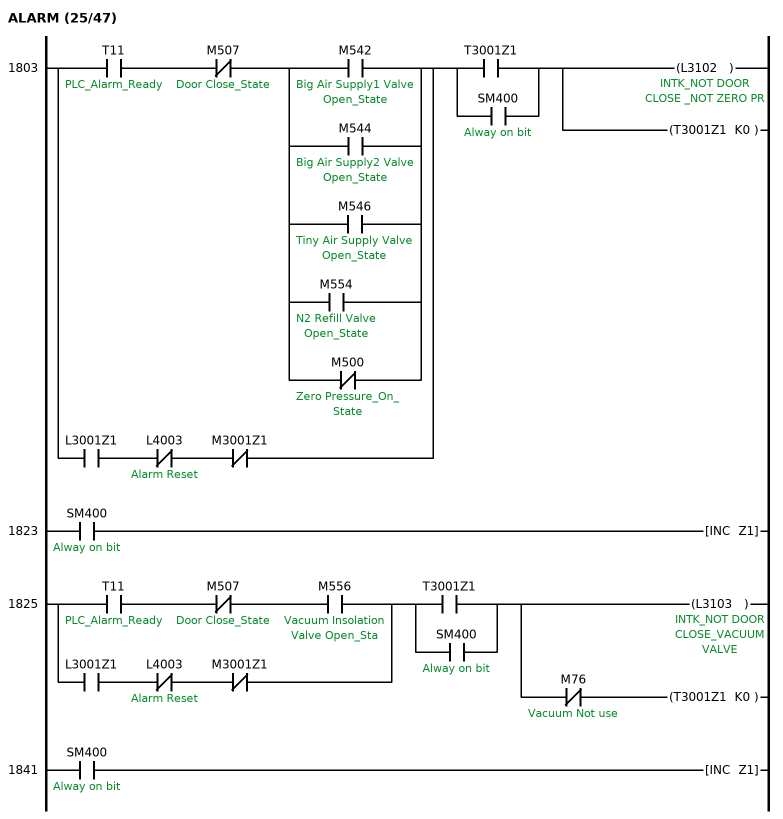
1803  LD      T11  ; PLC_Alarm_Ready
      ANI     M507  ; Door Close_State
      LD      M542  ; Big Air Supply1 Valve Open_State
      OR      M544  ; Big Air Supply2 Valve Open_State
      OR      M546  ; Tiny Air Supply Valve Open_State
      OR      M554  ; N2 Refill Valve Open_State
      ORI     M500  ; Zero Pressure_On_State
      ANB
      LD      L3001Z1
      ANI     L4003  ; Alarm Reset
      ANI     M3001Z1
      ORB
      LD      T3001Z1
      OR      SM400  ; Alway on bit
      ANB
      OUT     L3102  ; INTK_NOT DOOR CLOSE _NOT ZERO PR
      OUT     T3001Z1 K0
1823  LD      SM400  ; Alway on bit
      INC     Z1
1825  LD      T11  ; PLC_Alarm_Ready
      ANI     M507  ; Door Close_State
      AND     M556  ; Vacuum Insolation Valve Open_Sta
      LD      L3001Z1
      ANI     L4003  ; Alarm Reset
      ANI     M3001Z1
      ORB
      LD      T3001Z1
      OR      SM400  ; Alway on bit
      ANB
      OUT     L3103  ; INTK_NOT DOOR CLOSE_VACUUM VALVE
      ANI     M76  ; Vacuum Not use
      OUT     T3001Z1 K0
1841  LD      SM400  ; Alway on bit
      INC     Z1
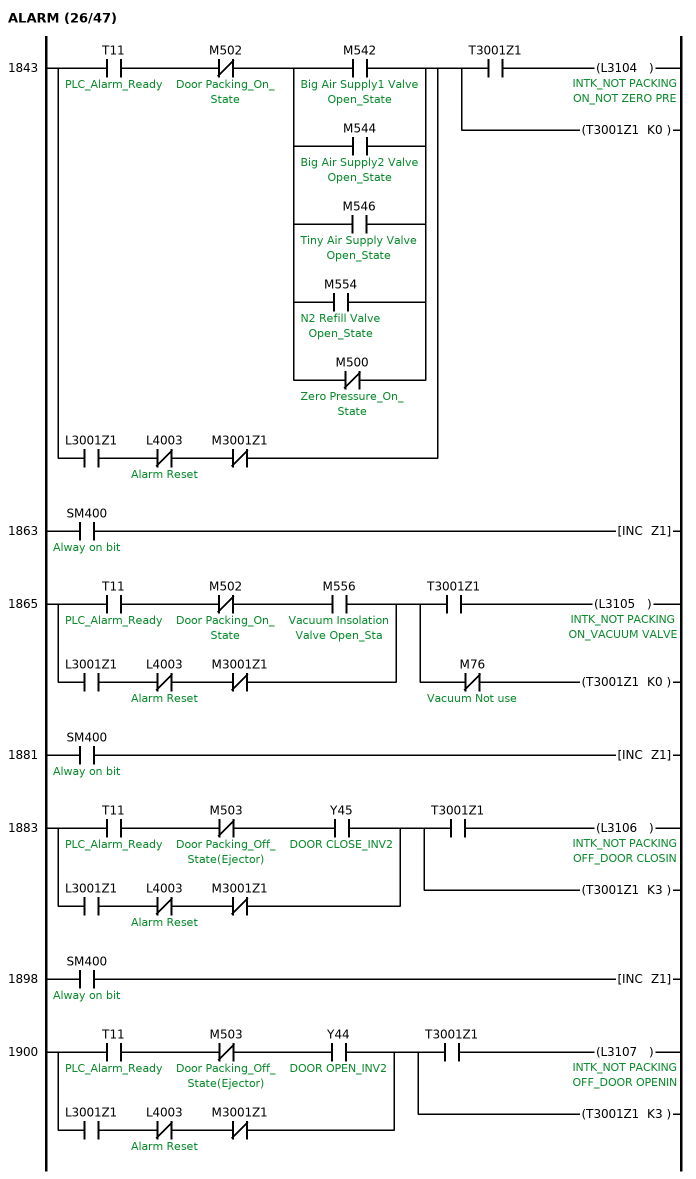
1843  LD      T11  ; PLC_Alarm_Ready
      ANI     M502  ; Door Packing_On_State
      LD      M542  ; Big Air Supply1 Valve Open_State
      OR      M544  ; Big Air Supply2 Valve Open_State
      OR      M546  ; Tiny Air Supply Valve Open_State
      OR      M554  ; N2 Refill Valve Open_State
      ORI     M500  ; Zero Pressure_On_State
      ANB
      LD      L3001Z1
      ANI     L4003  ; Alarm Reset
      ANI     M3001Z1
      ORB
      MPS
      AND     T3001Z1
      OUT     L3104  ; INTK_NOT PACKING ON_NOT ZERO PRE
      MPP
      OUT     T3001Z1 K0
1863  LD      SM400  ; Alway on bit
      INC     Z1
1865  LD      T11  ; PLC_Alarm_Ready
      ANI     M502  ; Door Packing_On_State
      AND     M556  ; Vacuum Insolation Valve Open_Sta
      LD      L3001Z1
      ANI     L4003  ; Alarm Reset
      ANI     M3001Z1
      ORB
      MPS
      AND     T3001Z1
      OUT     L3105  ; INTK_NOT PACKING ON_VACUUM VALVE
      MPP
      ANI     M76  ; Vacuum Not use
      OUT     T3001Z1 K0
1881  LD      SM400  ; Alway on bit
      INC     Z1
1883  LD      T11  ; PLC_Alarm_Ready
      ANI     M503  ; Door Packing_Off_State(Ejector)
      AND     Y45  ; DOOR CLOSE_INV2
      LD      L3001Z1
      ANI     L4003  ; Alarm Reset
      ANI     M3001Z1
      ORB
      MPS
      AND     T3001Z1
      OUT     L3106  ; INTK_NOT PACKING OFF_DOOR CLOSIN
      MPP
      OUT     T3001Z1 K3
1898  LD      SM400  ; Alway on bit
      INC     Z1
1900  LD      T11  ; PLC_Alarm_Ready
      ANI     M503  ; Door Packing_Off_State(Ejector)
      AND     Y44  ; DOOR OPEN_INV2
      LD      L3001Z1
      ANI     L4003  ; Alarm Reset
      ANI     M3001Z1
      ORB
      MPS
      AND     T3001Z1
      OUT     L3107  ; INTK_NOT PACKING OFF_DOOR OPENIN
      MPP
      OUT     T3001Z1 K3
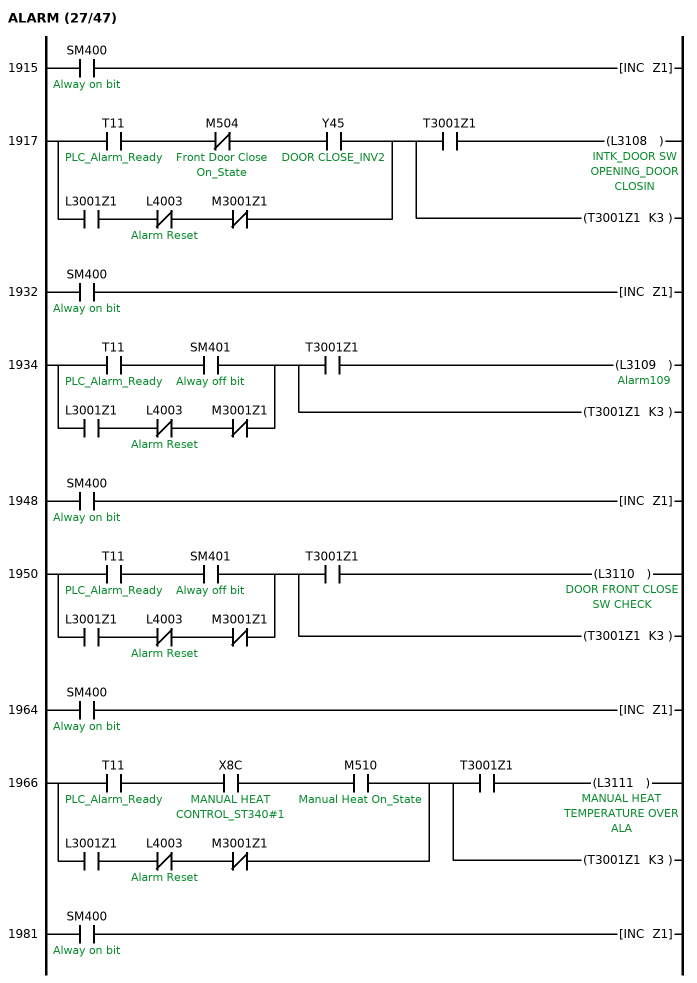
1915  LD      SM400  ; Alway on bit
      INC     Z1
1917  LD      T11  ; PLC_Alarm_Ready
      ANI     M504  ; Front Door Close On_State
      AND     Y45  ; DOOR CLOSE_INV2
      LD      L3001Z1
      ANI     L4003  ; Alarm Reset
      ANI     M3001Z1
      ORB
      MPS
      AND     T3001Z1
      OUT     L3108  ; INTK_DOOR SW OPENING_DOOR CLOSIN
      MPP
      OUT     T3001Z1 K3
1932  LD      SM400  ; Alway on bit
      INC     Z1
1934  LD      T11  ; PLC_Alarm_Ready
      AND     SM401  ; Alway off bit
      LD      L3001Z1
      ANI     L4003  ; Alarm Reset
      ANI     M3001Z1
      ORB
      MPS
      AND     T3001Z1
      OUT     L3109  ; Alarm109
      MPP
      OUT     T3001Z1 K3
1948  LD      SM400  ; Alway on bit
      INC     Z1
1950  LD      T11  ; PLC_Alarm_Ready
      AND     SM401  ; Alway off bit
      LD      L3001Z1
      ANI     L4003  ; Alarm Reset
      ANI     M3001Z1
      ORB
      MPS
      AND     T3001Z1
      OUT     L3110  ; DOOR FRONT CLOSE SW CHECK
      MPP
      OUT     T3001Z1 K3
1964  LD      SM400  ; Alway on bit
      INC     Z1
1966  LD      T11  ; PLC_Alarm_Ready
      AND     X8C  ; MANUAL HEAT CONTROL_ST340#1
      AND     M510  ; Manual Heat On_State
      LD      L3001Z1
      ANI     L4003  ; Alarm Reset
      ANI     M3001Z1
      ORB
      MPS
      AND     T3001Z1
      OUT     L3111  ; MANUAL HEAT TEMPERATURE OVER ALA
      MPP
      OUT     T3001Z1 K3
1981  LD      SM400  ; Alway on bit
      INC     Z1
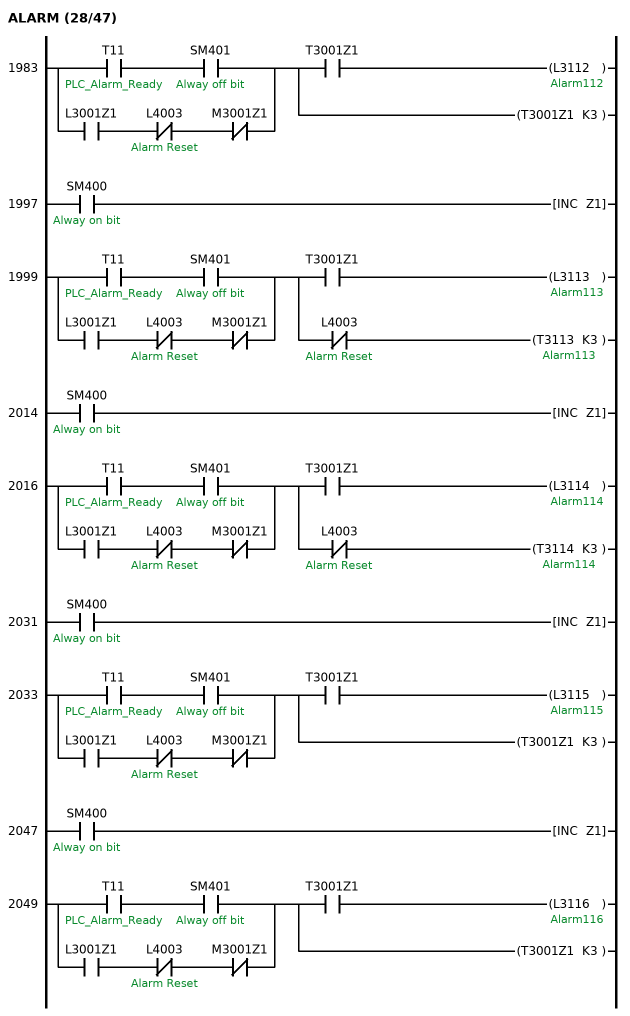
1983  LD      T11  ; PLC_Alarm_Ready
      AND     SM401  ; Alway off bit
      LD      L3001Z1
      ANI     L4003  ; Alarm Reset
      ANI     M3001Z1
      ORB
      MPS
      AND     T3001Z1
      OUT     L3112  ; Alarm112
      MPP
      OUT     T3001Z1 K3
1997  LD      SM400  ; Alway on bit
      INC     Z1
1999  LD      T11  ; PLC_Alarm_Ready
      AND     SM401  ; Alway off bit
      LD      L3001Z1
      ANI     L4003  ; Alarm Reset
      ANI     M3001Z1
      ORB
      MPS
      AND     T3001Z1
      OUT     L3113  ; Alarm113
      MPP
      ANI     L4003  ; Alarm Reset
      OUT     T3113 K3  ; Alarm113
2014  LD      SM400  ; Alway on bit
      INC     Z1
2016  LD      T11  ; PLC_Alarm_Ready
      AND     SM401  ; Alway off bit
      LD      L3001Z1
      ANI     L4003  ; Alarm Reset
      ANI     M3001Z1
      ORB
      MPS
      AND     T3001Z1
      OUT     L3114  ; Alarm114
      MPP
      ANI     L4003  ; Alarm Reset
      OUT     T3114 K3  ; Alarm114
2031  LD      SM400  ; Alway on bit
      INC     Z1
2033  LD      T11  ; PLC_Alarm_Ready
      AND     SM401  ; Alway off bit
      LD      L3001Z1
      ANI     L4003  ; Alarm Reset
      ANI     M3001Z1
      ORB
      MPS
      AND     T3001Z1
      OUT     L3115  ; Alarm115
      MPP
      OUT     T3001Z1 K3
2047  LD      SM400  ; Alway on bit
      INC     Z1
2049  LD      T11  ; PLC_Alarm_Ready
      AND     SM401  ; Alway off bit
      LD      L3001Z1
      ANI     L4003  ; Alarm Reset
      ANI     M3001Z1
      ORB
      MPS
      AND     T3001Z1
      OUT     L3116  ; Alarm116
      MPP
      OUT     T3001Z1 K3
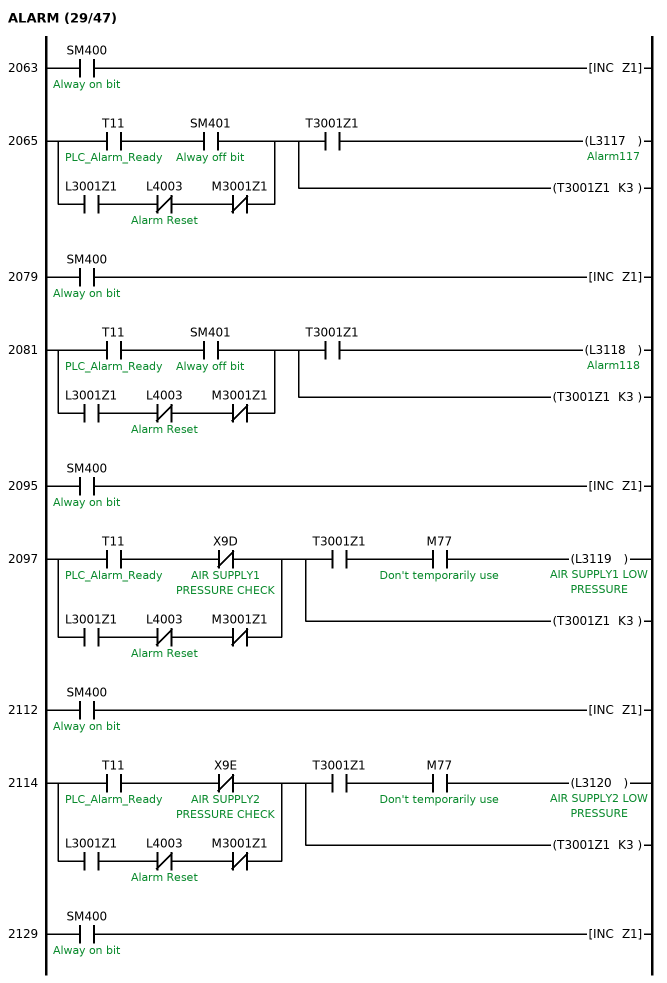
2063  LD      SM400  ; Alway on bit
      INC     Z1
2065  LD      T11  ; PLC_Alarm_Ready
      AND     SM401  ; Alway off bit
      LD      L3001Z1
      ANI     L4003  ; Alarm Reset
      ANI     M3001Z1
      ORB
      MPS
      AND     T3001Z1
      OUT     L3117  ; Alarm117
      MPP
      OUT     T3001Z1 K3
2079  LD      SM400  ; Alway on bit
      INC     Z1
2081  LD      T11  ; PLC_Alarm_Ready
      AND     SM401  ; Alway off bit
      LD      L3001Z1
      ANI     L4003  ; Alarm Reset
      ANI     M3001Z1
      ORB
      MPS
      AND     T3001Z1
      OUT     L3118  ; Alarm118
      MPP
      OUT     T3001Z1 K3
2095  LD      SM400  ; Alway on bit
      INC     Z1
2097  LD      T11  ; PLC_Alarm_Ready
      ANI     X9D  ; AIR SUPPLY1 PRESSURE CHECK
      LD      L3001Z1
      ANI     L4003  ; Alarm Reset
      ANI     M3001Z1
      ORB
      MPS
      AND     T3001Z1
      AND     M77  ; Don't temporarily use
      OUT     L3119  ; AIR SUPPLY1 LOW PRESSURE
      MPP
      OUT     T3001Z1 K3
2112  LD      SM400  ; Alway on bit
      INC     Z1
2114  LD      T11  ; PLC_Alarm_Ready
      ANI     X9E  ; AIR SUPPLY2 PRESSURE CHECK
      LD      L3001Z1
      ANI     L4003  ; Alarm Reset
      ANI     M3001Z1
      ORB
      MPS
      AND     T3001Z1
      AND     M77  ; Don't temporarily use
      OUT     L3120  ; AIR SUPPLY2 LOW PRESSURE
      MPP
      OUT     T3001Z1 K3
2129  LD      SM400  ; Alway on bit
      INC     Z1
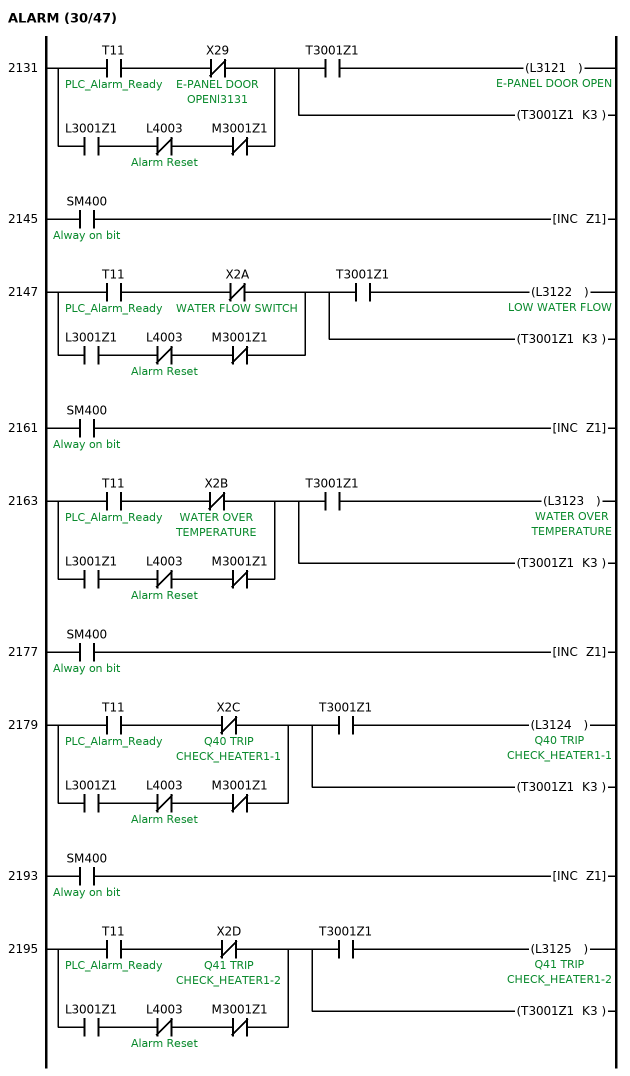
2131  LD      T11  ; PLC_Alarm_Ready
      ANI     X29  ; E-PANEL DOOR OPENl3131
      LD      L3001Z1
      ANI     L4003  ; Alarm Reset
      ANI     M3001Z1
      ORB
      MPS
      AND     T3001Z1
      OUT     L3121  ; E-PANEL DOOR OPEN
      MPP
      OUT     T3001Z1 K3
2145  LD      SM400  ; Alway on bit
      INC     Z1
2147  LD      T11  ; PLC_Alarm_Ready
      ANI     X2A  ; WATER FLOW SWITCH
      LD      L3001Z1
      ANI     L4003  ; Alarm Reset
      ANI     M3001Z1
      ORB
      MPS
      AND     T3001Z1
      OUT     L3122  ; LOW WATER FLOW
      MPP
      OUT     T3001Z1 K3
2161  LD      SM400  ; Alway on bit
      INC     Z1
2163  LD      T11  ; PLC_Alarm_Ready
      ANI     X2B  ; WATER OVER TEMPERATURE
      LD      L3001Z1
      ANI     L4003  ; Alarm Reset
      ANI     M3001Z1
      ORB
      MPS
      AND     T3001Z1
      OUT     L3123  ; WATER OVER TEMPERATURE
      MPP
      OUT     T3001Z1 K3
2177  LD      SM400  ; Alway on bit
      INC     Z1
2179  LD      T11  ; PLC_Alarm_Ready
      ANI     X2C  ; Q40 TRIP CHECK_HEATER1-1
      LD      L3001Z1
      ANI     L4003  ; Alarm Reset
      ANI     M3001Z1
      ORB
      MPS
      AND     T3001Z1
      OUT     L3124  ; Q40 TRIP CHECK_HEATER1-1
      MPP
      OUT     T3001Z1 K3
2193  LD      SM400  ; Alway on bit
      INC     Z1
2195  LD      T11  ; PLC_Alarm_Ready
      ANI     X2D  ; Q41 TRIP CHECK_HEATER1-2
      LD      L3001Z1
      ANI     L4003  ; Alarm Reset
      ANI     M3001Z1
      ORB
      MPS
      AND     T3001Z1
      OUT     L3125  ; Q41 TRIP CHECK_HEATER1-2
      MPP
      OUT     T3001Z1 K3
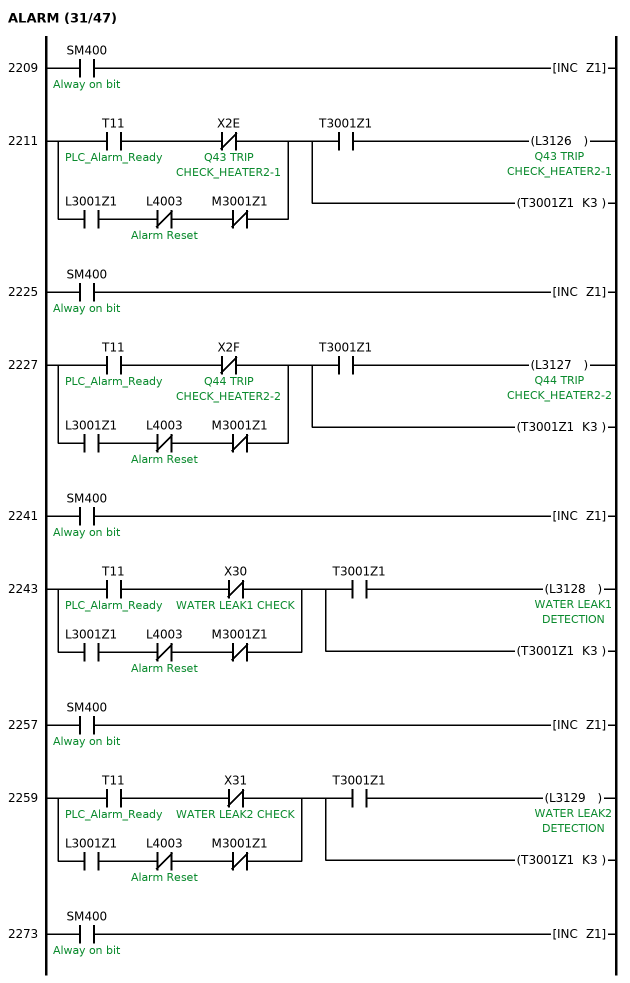
2209  LD      SM400  ; Alway on bit
      INC     Z1
2211  LD      T11  ; PLC_Alarm_Ready
      ANI     X2E  ; Q43 TRIP CHECK_HEATER2-1
      LD      L3001Z1
      ANI     L4003  ; Alarm Reset
      ANI     M3001Z1
      ORB
      MPS
      AND     T3001Z1
      OUT     L3126  ; Q43 TRIP CHECK_HEATER2-1
      MPP
      OUT     T3001Z1 K3
2225  LD      SM400  ; Alway on bit
      INC     Z1
2227  LD      T11  ; PLC_Alarm_Ready
      ANI     X2F  ; Q44 TRIP CHECK_HEATER2-2
      LD      L3001Z1
      ANI     L4003  ; Alarm Reset
      ANI     M3001Z1
      ORB
      MPS
      AND     T3001Z1
      OUT     L3127  ; Q44 TRIP CHECK_HEATER2-2
      MPP
      OUT     T3001Z1 K3
2241  LD      SM400  ; Alway on bit
      INC     Z1
2243  LD      T11  ; PLC_Alarm_Ready
      ANI     X30  ; WATER LEAK1 CHECK
      LD      L3001Z1
      ANI     L4003  ; Alarm Reset
      ANI     M3001Z1
      ORB
      MPS
      AND     T3001Z1
      OUT     L3128  ; WATER LEAK1 DETECTION
      MPP
      OUT     T3001Z1 K3
2257  LD      SM400  ; Alway on bit
      INC     Z1
2259  LD      T11  ; PLC_Alarm_Ready
      ANI     X31  ; WATER LEAK2 CHECK
      LD      L3001Z1
      ANI     L4003  ; Alarm Reset
      ANI     M3001Z1
      ORB
      MPS
      AND     T3001Z1
      OUT     L3129  ; WATER LEAK2 DETECTION
      MPP
      OUT     T3001Z1 K3
2273  LD      SM400  ; Alway on bit
      INC     Z1
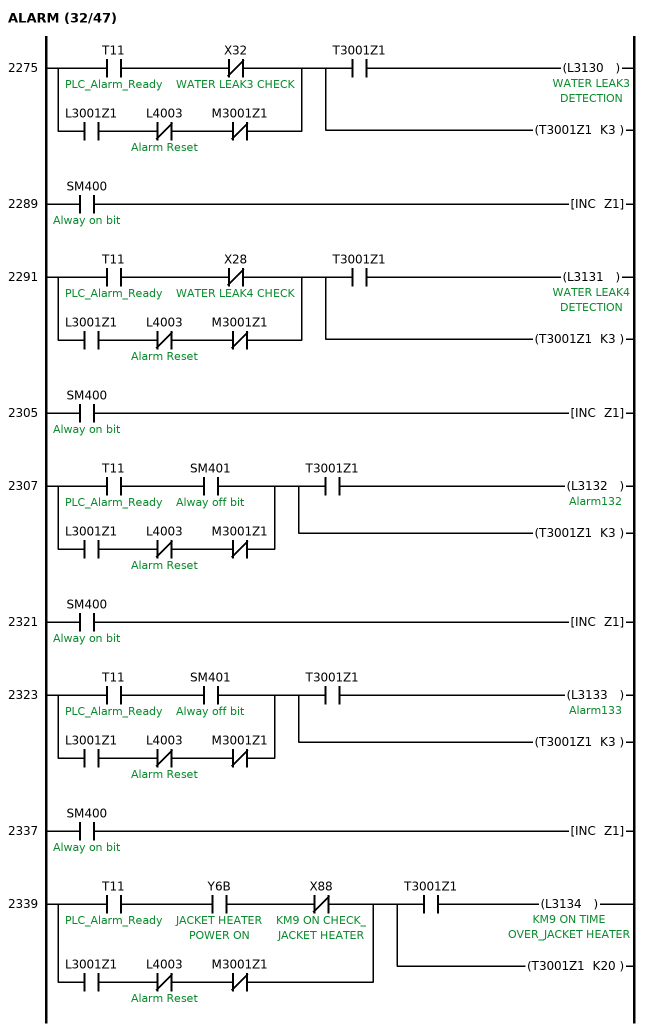
2275  LD      T11  ; PLC_Alarm_Ready
      ANI     X32  ; WATER LEAK3 CHECK
      LD      L3001Z1
      ANI     L4003  ; Alarm Reset
      ANI     M3001Z1
      ORB
      MPS
      AND     T3001Z1
      OUT     L3130  ; WATER LEAK3 DETECTION
      MPP
      OUT     T3001Z1 K3
2289  LD      SM400  ; Alway on bit
      INC     Z1
2291  LD      T11  ; PLC_Alarm_Ready
      ANI     X28  ; WATER LEAK4 CHECK
      LD      L3001Z1
      ANI     L4003  ; Alarm Reset
      ANI     M3001Z1
      ORB
      MPS
      AND     T3001Z1
      OUT     L3131  ; WATER LEAK4 DETECTION
      MPP
      OUT     T3001Z1 K3
2305  LD      SM400  ; Alway on bit
      INC     Z1
2307  LD      T11  ; PLC_Alarm_Ready
      AND     SM401  ; Alway off bit
      LD      L3001Z1
      ANI     L4003  ; Alarm Reset
      ANI     M3001Z1
      ORB
      MPS
      AND     T3001Z1
      OUT     L3132  ; Alarm132
      MPP
      OUT     T3001Z1 K3
2321  LD      SM400  ; Alway on bit
      INC     Z1
2323  LD      T11  ; PLC_Alarm_Ready
      AND     SM401  ; Alway off bit
      LD      L3001Z1
      ANI     L4003  ; Alarm Reset
      ANI     M3001Z1
      ORB
      MPS
      AND     T3001Z1
      OUT     L3133  ; Alarm133
      MPP
      OUT     T3001Z1 K3
2337  LD      SM400  ; Alway on bit
      INC     Z1
2339  LD      T11  ; PLC_Alarm_Ready
      AND     Y6B  ; JACKET HEATER POWER ON
      ANI     X88  ; KM9 ON CHECK_JACKET HEATER
      LD      L3001Z1
      ANI     L4003  ; Alarm Reset
      ANI     M3001Z1
      ORB
      MPS
      AND     T3001Z1
      OUT     L3134  ; KM9 ON TIME OVER_JACKET HEATER
      MPP
      OUT     T3001Z1 K20
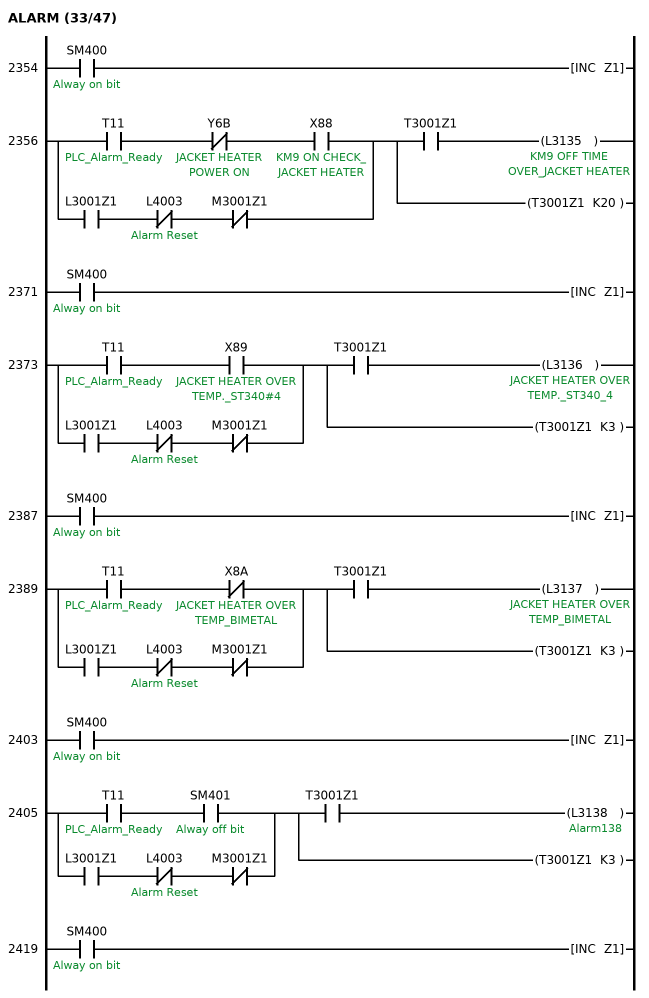
2354  LD      SM400  ; Alway on bit
      INC     Z1
2356  LD      T11  ; PLC_Alarm_Ready
      ANI     Y6B  ; JACKET HEATER POWER ON
      AND     X88  ; KM9 ON CHECK_JACKET HEATER
      LD      L3001Z1
      ANI     L4003  ; Alarm Reset
      ANI     M3001Z1
      ORB
      MPS
      AND     T3001Z1
      OUT     L3135  ; KM9 OFF TIME OVER_JACKET HEATER
      MPP
      OUT     T3001Z1 K20
2371  LD      SM400  ; Alway on bit
      INC     Z1
2373  LD      T11  ; PLC_Alarm_Ready
      AND     X89  ; JACKET HEATER OVER TEMP._ST340#4
      LD      L3001Z1
      ANI     L4003  ; Alarm Reset
      ANI     M3001Z1
      ORB
      MPS
      AND     T3001Z1
      OUT     L3136  ; JACKET HEATER OVER TEMP._ST340_4
      MPP
      OUT     T3001Z1 K3
2387  LD      SM400  ; Alway on bit
      INC     Z1
2389  LD      T11  ; PLC_Alarm_Ready
      ANI     X8A  ; JACKET HEATER OVER TEMP_BIMETAL
      LD      L3001Z1
      ANI     L4003  ; Alarm Reset
      ANI     M3001Z1
      ORB
      MPS
      AND     T3001Z1
      OUT     L3137  ; JACKET HEATER OVER TEMP_BIMETAL
      MPP
      OUT     T3001Z1 K3
2403  LD      SM400  ; Alway on bit
      INC     Z1
2405  LD      T11  ; PLC_Alarm_Ready
      AND     SM401  ; Alway off bit
      LD      L3001Z1
      ANI     L4003  ; Alarm Reset
      ANI     M3001Z1
      ORB
      MPS
      AND     T3001Z1
      OUT     L3138  ; Alarm138
      MPP
      OUT     T3001Z1 K3
2419  LD      SM400  ; Alway on bit
      INC     Z1
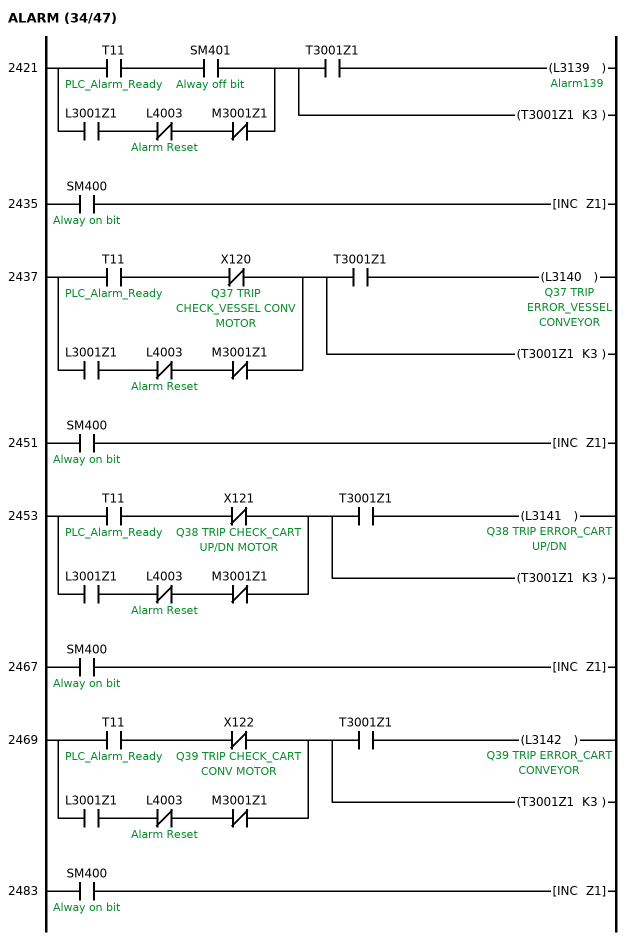
2421  LD      T11  ; PLC_Alarm_Ready
      AND     SM401  ; Alway off bit
      LD      L3001Z1
      ANI     L4003  ; Alarm Reset
      ANI     M3001Z1
      ORB
      MPS
      AND     T3001Z1
      OUT     L3139  ; Alarm139
      MPP
      OUT     T3001Z1 K3
2435  LD      SM400  ; Alway on bit
      INC     Z1
2437  LD      T11  ; PLC_Alarm_Ready
      ANI     X120  ; Q37 TRIP CHECK_VESSEL CONV MOTOR
      LD      L3001Z1
      ANI     L4003  ; Alarm Reset
      ANI     M3001Z1
      ORB
      MPS
      AND     T3001Z1
      OUT     L3140  ; Q37 TRIP ERROR_VESSEL CONVEYOR
      MPP
      OUT     T3001Z1 K3
2451  LD      SM400  ; Alway on bit
      INC     Z1
2453  LD      T11  ; PLC_Alarm_Ready
      ANI     X121  ; Q38 TRIP CHECK_CART UP/DN MOTOR
      LD      L3001Z1
      ANI     L4003  ; Alarm Reset
      ANI     M3001Z1
      ORB
      MPS
      AND     T3001Z1
      OUT     L3141  ; Q38 TRIP ERROR_CART UP/DN
      MPP
      OUT     T3001Z1 K3
2467  LD      SM400  ; Alway on bit
      INC     Z1
2469  LD      T11  ; PLC_Alarm_Ready
      ANI     X122  ; Q39 TRIP CHECK_CART CONV MOTOR
      LD      L3001Z1
      ANI     L4003  ; Alarm Reset
      ANI     M3001Z1
      ORB
      MPS
      AND     T3001Z1
      OUT     L3142  ; Q39 TRIP ERROR_CART CONVEYOR
      MPP
      OUT     T3001Z1 K3
2483  LD      SM400  ; Alway on bit
      INC     Z1
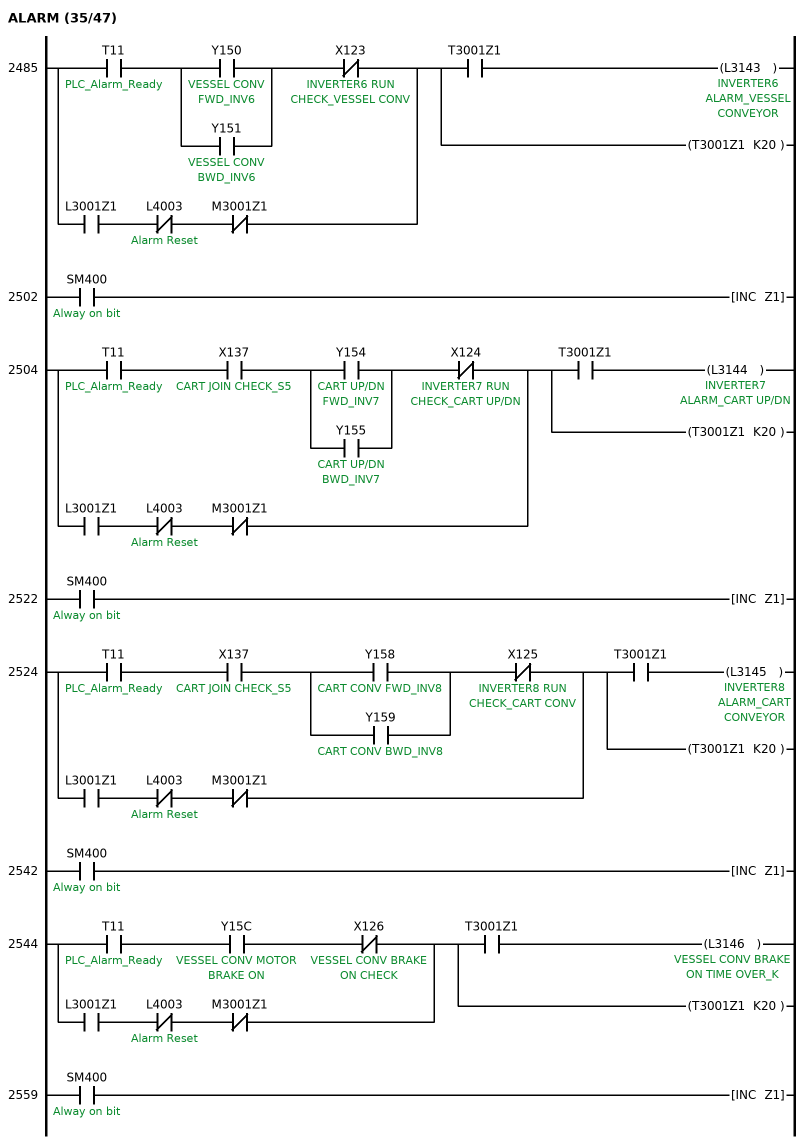
2485  LD      T11  ; PLC_Alarm_Ready
      LD      Y150  ; VESSEL CONV FWD_INV6
      OR      Y151  ; VESSEL CONV BWD_INV6
      ANB
      ANI     X123  ; INVERTER6 RUN CHECK_VESSEL CONV
      LD      L3001Z1
      ANI     L4003  ; Alarm Reset
      ANI     M3001Z1
      ORB
      MPS
      AND     T3001Z1
      OUT     L3143  ; INVERTER6 ALARM_VESSEL CONVEYOR
      MPP
      OUT     T3001Z1 K20
2502  LD      SM400  ; Alway on bit
      INC     Z1
2504  LD      T11  ; PLC_Alarm_Ready
      AND     X137  ; CART JOIN CHECK_S5
      LD      Y154  ; CART UP/DN FWD_INV7
      OR      Y155  ; CART UP/DN BWD_INV7
      ANB
      ANI     X124  ; INVERTER7 RUN CHECK_CART UP/DN
      LD      L3001Z1
      ANI     L4003  ; Alarm Reset
      ANI     M3001Z1
      ORB
      MPS
      AND     T3001Z1
      OUT     L3144  ; INVERTER7 ALARM_CART UP/DN
      MPP
      OUT     T3001Z1 K20
2522  LD      SM400  ; Alway on bit
      INC     Z1
2524  LD      T11  ; PLC_Alarm_Ready
      AND     X137  ; CART JOIN CHECK_S5
      LD      Y158  ; CART CONV FWD_INV8
      OR      Y159  ; CART CONV BWD_INV8
      ANB
      ANI     X125  ; INVERTER8 RUN CHECK_CART CONV
      LD      L3001Z1
      ANI     L4003  ; Alarm Reset
      ANI     M3001Z1
      ORB
      MPS
      AND     T3001Z1
      OUT     L3145  ; INVERTER8 ALARM_CART CONVEYOR
      MPP
      OUT     T3001Z1 K20
2542  LD      SM400  ; Alway on bit
      INC     Z1
2544  LD      T11  ; PLC_Alarm_Ready
      AND     Y15C  ; VESSEL CONV MOTOR BRAKE ON
      ANI     X126  ; VESSEL CONV BRAKE ON CHECK
      LD      L3001Z1
      ANI     L4003  ; Alarm Reset
      ANI     M3001Z1
      ORB
      MPS
      AND     T3001Z1
      OUT     L3146  ; VESSEL CONV BRAKE ON TIME OVER_K
      MPP
      OUT     T3001Z1 K20
2559  LD      SM400  ; Alway on bit
      INC     Z1
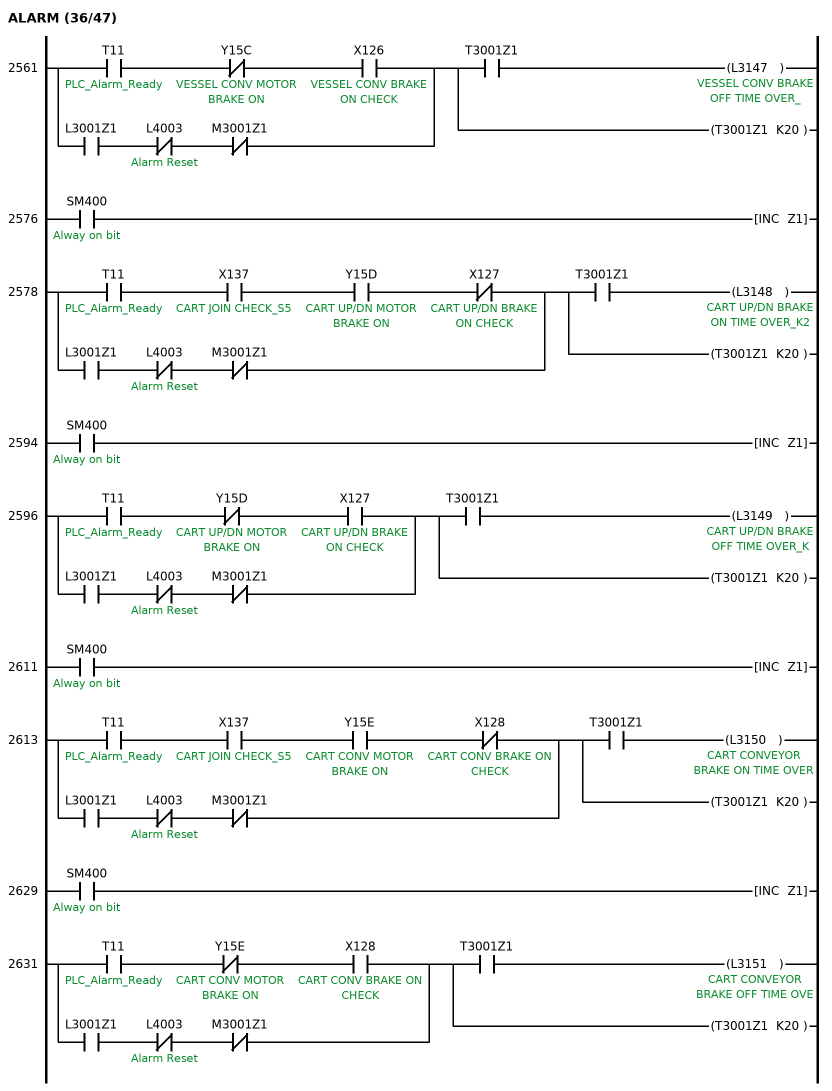
2561  LD      T11  ; PLC_Alarm_Ready
      ANI     Y15C  ; VESSEL CONV MOTOR BRAKE ON
      AND     X126  ; VESSEL CONV BRAKE ON CHECK
      LD      L3001Z1
      ANI     L4003  ; Alarm Reset
      ANI     M3001Z1
      ORB
      MPS
      AND     T3001Z1
      OUT     L3147  ; VESSEL CONV BRAKE OFF TIME OVER_
      MPP
      OUT     T3001Z1 K20
2576  LD      SM400  ; Alway on bit
      INC     Z1
2578  LD      T11  ; PLC_Alarm_Ready
      AND     X137  ; CART JOIN CHECK_S5
      AND     Y15D  ; CART UP/DN MOTOR BRAKE ON
      ANI     X127  ; CART UP/DN BRAKE ON CHECK
      LD      L3001Z1
      ANI     L4003  ; Alarm Reset
      ANI     M3001Z1
      ORB
      MPS
      AND     T3001Z1
      OUT     L3148  ; CART UP/DN BRAKE ON TIME OVER_K2
      MPP
      OUT     T3001Z1 K20
2594  LD      SM400  ; Alway on bit
      INC     Z1
2596  LD      T11  ; PLC_Alarm_Ready
      ANI     Y15D  ; CART UP/DN MOTOR BRAKE ON
      AND     X127  ; CART UP/DN BRAKE ON CHECK
      LD      L3001Z1
      ANI     L4003  ; Alarm Reset
      ANI     M3001Z1
      ORB
      MPS
      AND     T3001Z1
      OUT     L3149  ; CART UP/DN BRAKE OFF TIME OVER_K
      MPP
      OUT     T3001Z1 K20
2611  LD      SM400  ; Alway on bit
      INC     Z1
2613  LD      T11  ; PLC_Alarm_Ready
      AND     X137  ; CART JOIN CHECK_S5
      AND     Y15E  ; CART CONV MOTOR BRAKE ON
      ANI     X128  ; CART CONV BRAKE ON CHECK
      LD      L3001Z1
      ANI     L4003  ; Alarm Reset
      ANI     M3001Z1
      ORB
      MPS
      AND     T3001Z1
      OUT     L3150  ; CART CONVEYOR BRAKE ON TIME OVER
      MPP
      OUT     T3001Z1 K20
2629  LD      SM400  ; Alway on bit
      INC     Z1
2631  LD      T11  ; PLC_Alarm_Ready
      ANI     Y15E  ; CART CONV MOTOR BRAKE ON
      AND     X128  ; CART CONV BRAKE ON CHECK
      LD      L3001Z1
      ANI     L4003  ; Alarm Reset
      ANI     M3001Z1
      ORB
      MPS
      AND     T3001Z1
      OUT     L3151  ; CART CONVEYOR BRAKE OFF TIME OVE
      MPP
      OUT     T3001Z1 K20
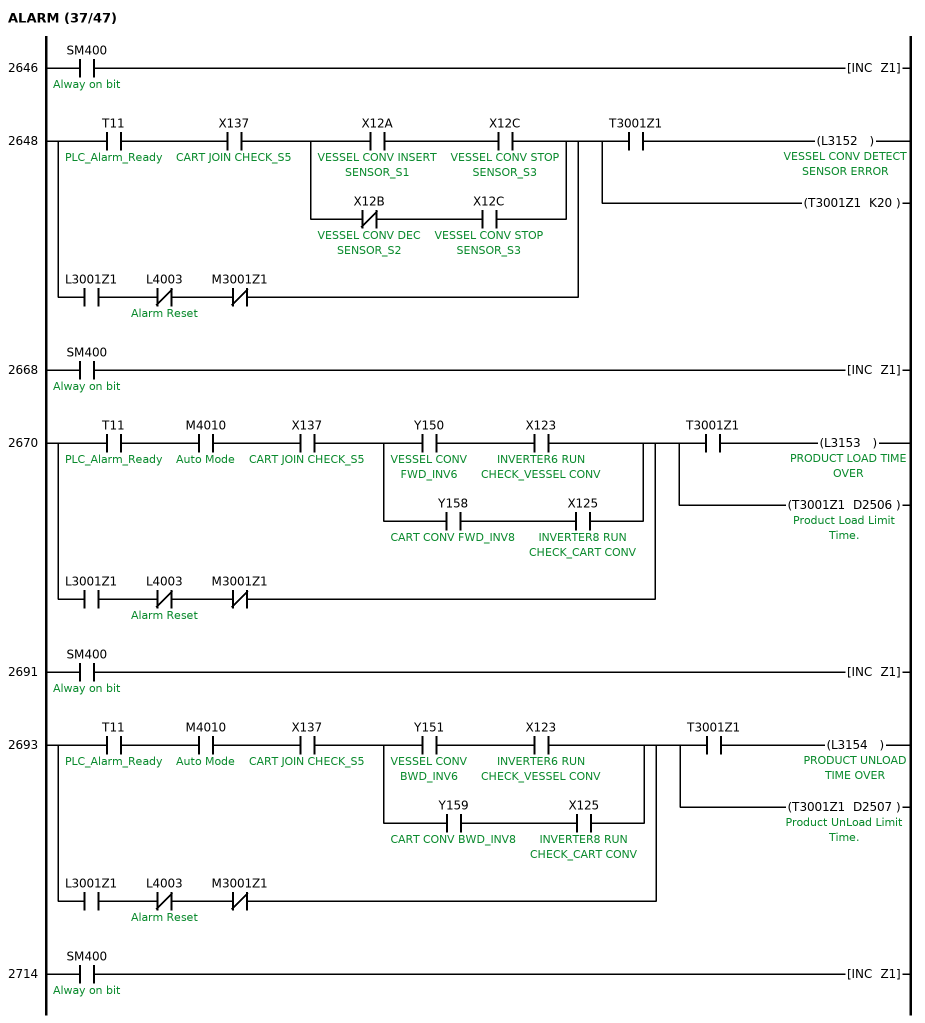
2646  LD      SM400  ; Alway on bit
      INC     Z1
2648  LD      T11  ; PLC_Alarm_Ready
      AND     X137  ; CART JOIN CHECK_S5
      LD      X12A  ; VESSEL CONV INSERT SENSOR_S1
      AND     X12C  ; VESSEL CONV STOP SENSOR_S3
      LDI     X12B  ; VESSEL CONV DEC SENSOR_S2
      AND     X12C  ; VESSEL CONV STOP SENSOR_S3
      ORB
      ANB
      LD      L3001Z1
      ANI     L4003  ; Alarm Reset
      ANI     M3001Z1
      ORB
      MPS
      AND     T3001Z1
      OUT     L3152  ; VESSEL CONV DETECT SENSOR ERROR
      MPP
      OUT     T3001Z1 K20
2668  LD      SM400  ; Alway on bit
      INC     Z1
2670  LD      T11  ; PLC_Alarm_Ready
      AND     M4010  ; Auto Mode
      AND     X137  ; CART JOIN CHECK_S5
      LD      Y150  ; VESSEL CONV FWD_INV6
      AND     X123  ; INVERTER6 RUN CHECK_VESSEL CONV
      LD      Y158  ; CART CONV FWD_INV8
      AND     X125  ; INVERTER8 RUN CHECK_CART CONV
      ORB
      ANB
      LD      L3001Z1
      ANI     L4003  ; Alarm Reset
      ANI     M3001Z1
      ORB
      MPS
      AND     T3001Z1
      OUT     L3153  ; PRODUCT LOAD TIME OVER
      MPP
      OUT     T3001Z1 D2506  ; Product Load Limit Time.
2691  LD      SM400  ; Alway on bit
      INC     Z1
2693  LD      T11  ; PLC_Alarm_Ready
      AND     M4010  ; Auto Mode
      AND     X137  ; CART JOIN CHECK_S5
      LD      Y151  ; VESSEL CONV BWD_INV6
      AND     X123  ; INVERTER6 RUN CHECK_VESSEL CONV
      LD      Y159  ; CART CONV BWD_INV8
      AND     X125  ; INVERTER8 RUN CHECK_CART CONV
      ORB
      ANB
      LD      L3001Z1
      ANI     L4003  ; Alarm Reset
      ANI     M3001Z1
      ORB
      MPS
      AND     T3001Z1
      OUT     L3154  ; PRODUCT UNLOAD TIME OVER
      MPP
      OUT     T3001Z1 D2507  ; Product UnLoad Limit Time.
2714  LD      SM400  ; Alway on bit
      INC     Z1
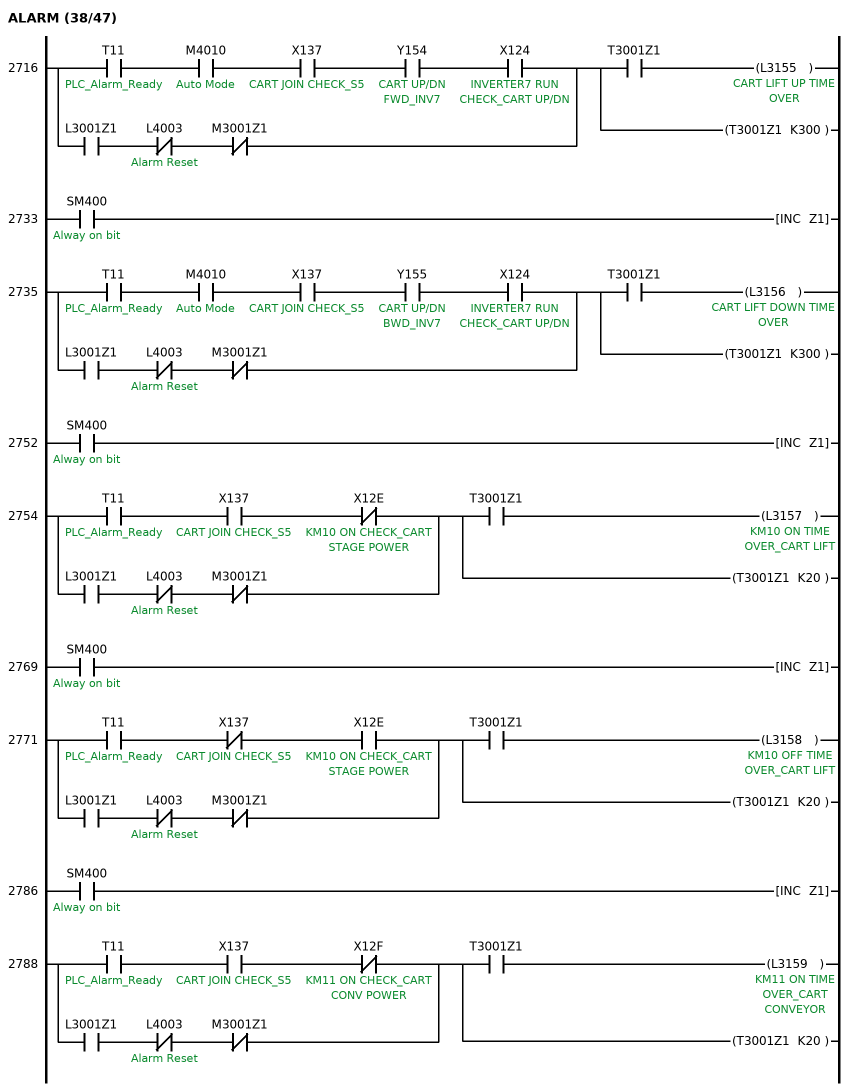
2716  LD      T11  ; PLC_Alarm_Ready
      AND     M4010  ; Auto Mode
      AND     X137  ; CART JOIN CHECK_S5
      AND     Y154  ; CART UP/DN FWD_INV7
      AND     X124  ; INVERTER7 RUN CHECK_CART UP/DN
      LD      L3001Z1
      ANI     L4003  ; Alarm Reset
      ANI     M3001Z1
      ORB
      MPS
      AND     T3001Z1
      OUT     L3155  ; CART LIFT UP TIME OVER
      MPP
      OUT     T3001Z1 K300
2733  LD      SM400  ; Alway on bit
      INC     Z1
2735  LD      T11  ; PLC_Alarm_Ready
      AND     M4010  ; Auto Mode
      AND     X137  ; CART JOIN CHECK_S5
      AND     Y155  ; CART UP/DN BWD_INV7
      AND     X124  ; INVERTER7 RUN CHECK_CART UP/DN
      LD      L3001Z1
      ANI     L4003  ; Alarm Reset
      ANI     M3001Z1
      ORB
      MPS
      AND     T3001Z1
      OUT     L3156  ; CART LIFT DOWN TIME OVER
      MPP
      OUT     T3001Z1 K300
2752  LD      SM400  ; Alway on bit
      INC     Z1
2754  LD      T11  ; PLC_Alarm_Ready
      AND     X137  ; CART JOIN CHECK_S5
      ANI     X12E  ; KM10 ON CHECK_CART STAGE POWER
      LD      L3001Z1
      ANI     L4003  ; Alarm Reset
      ANI     M3001Z1
      ORB
      MPS
      AND     T3001Z1
      OUT     L3157  ; KM10 ON TIME OVER_CART LIFT
      MPP
      OUT     T3001Z1 K20
2769  LD      SM400  ; Alway on bit
      INC     Z1
2771  LD      T11  ; PLC_Alarm_Ready
      ANI     X137  ; CART JOIN CHECK_S5
      AND     X12E  ; KM10 ON CHECK_CART STAGE POWER
      LD      L3001Z1
      ANI     L4003  ; Alarm Reset
      ANI     M3001Z1
      ORB
      MPS
      AND     T3001Z1
      OUT     L3158  ; KM10 OFF TIME OVER_CART LIFT
      MPP
      OUT     T3001Z1 K20
2786  LD      SM400  ; Alway on bit
      INC     Z1
2788  LD      T11  ; PLC_Alarm_Ready
      AND     X137  ; CART JOIN CHECK_S5
      ANI     X12F  ; KM11 ON CHECK_CART CONV POWER
      LD      L3001Z1
      ANI     L4003  ; Alarm Reset
      ANI     M3001Z1
      ORB
      MPS
      AND     T3001Z1
      OUT     L3159  ; KM11 ON TIME OVER_CART CONVEYOR
      MPP
      OUT     T3001Z1 K20
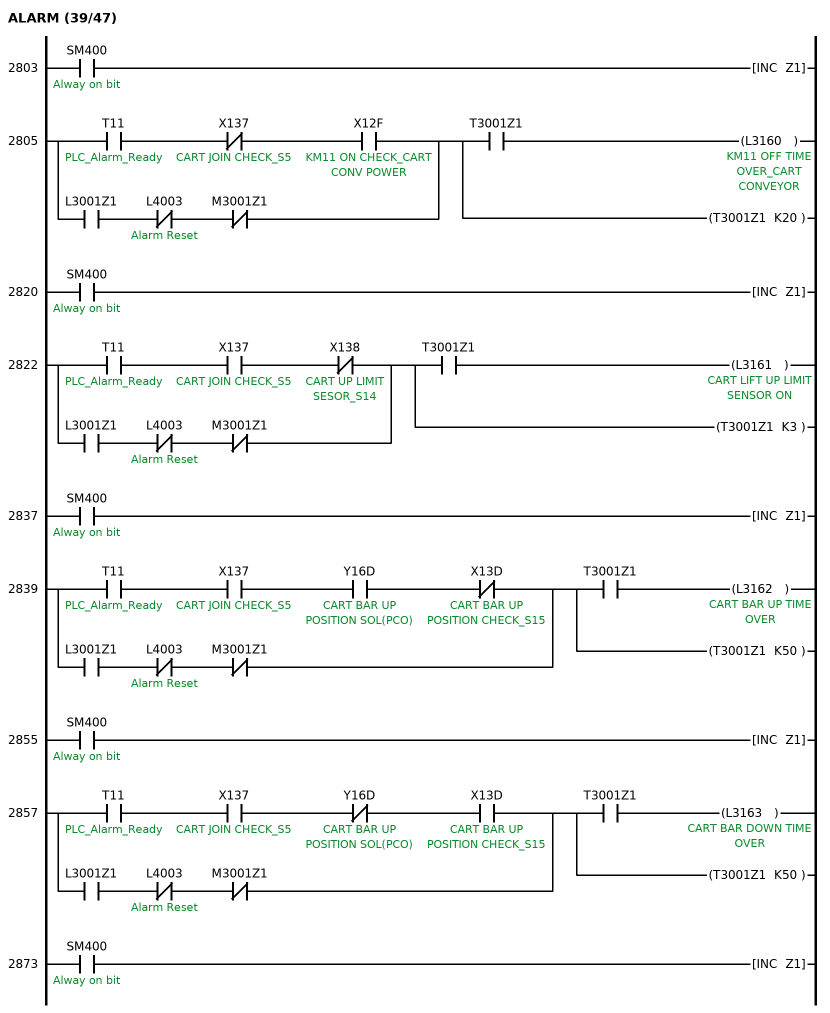
2803  LD      SM400  ; Alway on bit
      INC     Z1
2805  LD      T11  ; PLC_Alarm_Ready
      ANI     X137  ; CART JOIN CHECK_S5
      AND     X12F  ; KM11 ON CHECK_CART CONV POWER
      LD      L3001Z1
      ANI     L4003  ; Alarm Reset
      ANI     M3001Z1
      ORB
      MPS
      AND     T3001Z1
      OUT     L3160  ; KM11 OFF TIME OVER_CART CONVEYOR
      MPP
      OUT     T3001Z1 K20
2820  LD      SM400  ; Alway on bit
      INC     Z1
2822  LD      T11  ; PLC_Alarm_Ready
      AND     X137  ; CART JOIN CHECK_S5
      ANI     X138  ; CART UP LIMIT SESOR_S14
      LD      L3001Z1
      ANI     L4003  ; Alarm Reset
      ANI     M3001Z1
      ORB
      MPS
      AND     T3001Z1
      OUT     L3161  ; CART LIFT UP LIMIT SENSOR ON
      MPP
      OUT     T3001Z1 K3
2837  LD      SM400  ; Alway on bit
      INC     Z1
2839  LD      T11  ; PLC_Alarm_Ready
      AND     X137  ; CART JOIN CHECK_S5
      AND     Y16D  ; CART BAR UP POSITION SOL(PCO)
      ANI     X13D  ; CART BAR UP POSITION CHECK_S15
      LD      L3001Z1
      ANI     L4003  ; Alarm Reset
      ANI     M3001Z1
      ORB
      MPS
      AND     T3001Z1
      OUT     L3162  ; CART BAR UP TIME OVER
      MPP
      OUT     T3001Z1 K50
2855  LD      SM400  ; Alway on bit
      INC     Z1
2857  LD      T11  ; PLC_Alarm_Ready
      AND     X137  ; CART JOIN CHECK_S5
      ANI     Y16D  ; CART BAR UP POSITION SOL(PCO)
      AND     X13D  ; CART BAR UP POSITION CHECK_S15
      LD      L3001Z1
      ANI     L4003  ; Alarm Reset
      ANI     M3001Z1
      ORB
      MPS
      AND     T3001Z1
      OUT     L3163  ; CART BAR DOWN TIME OVER
      MPP
      OUT     T3001Z1 K50
2873  LD      SM400  ; Alway on bit
      INC     Z1
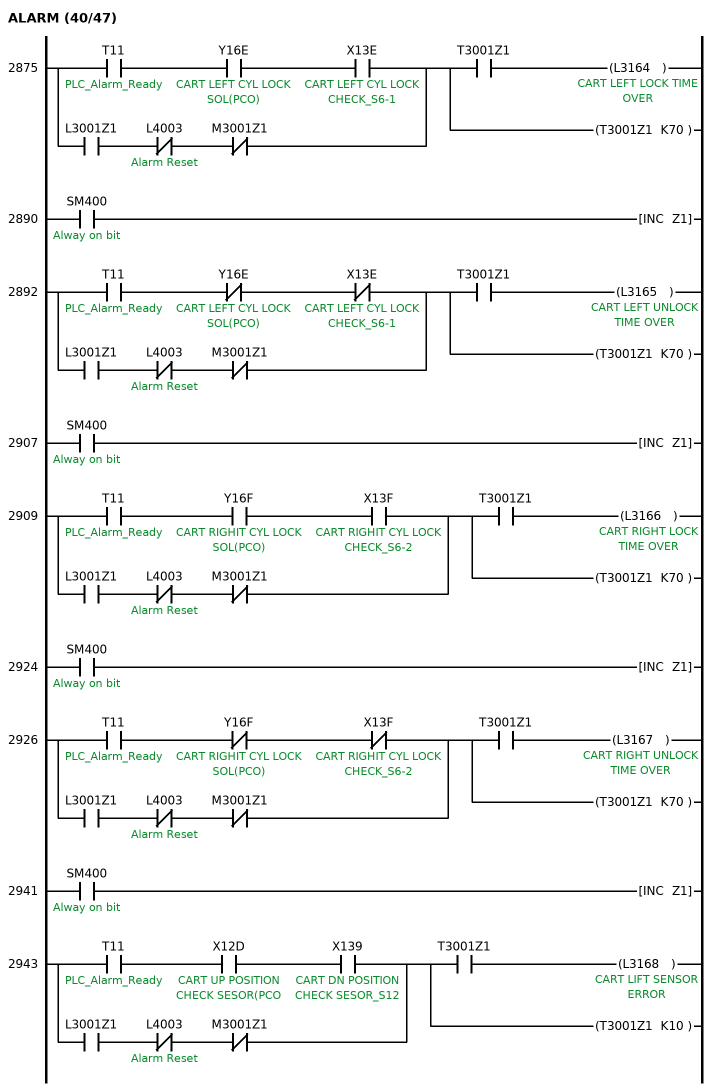
2875  LD      T11  ; PLC_Alarm_Ready
      AND     Y16E  ; CART LEFT CYL LOCK SOL(PCO)
      AND     X13E  ; CART LEFT CYL LOCK CHECK_S6-1
      LD      L3001Z1
      ANI     L4003  ; Alarm Reset
      ANI     M3001Z1
      ORB
      MPS
      AND     T3001Z1
      OUT     L3164  ; CART LEFT LOCK TIME OVER
      MPP
      OUT     T3001Z1 K70
2890  LD      SM400  ; Alway on bit
      INC     Z1
2892  LD      T11  ; PLC_Alarm_Ready
      ANI     Y16E  ; CART LEFT CYL LOCK SOL(PCO)
      ANI     X13E  ; CART LEFT CYL LOCK CHECK_S6-1
      LD      L3001Z1
      ANI     L4003  ; Alarm Reset
      ANI     M3001Z1
      ORB
      MPS
      AND     T3001Z1
      OUT     L3165  ; CART LEFT UNLOCK TIME OVER
      MPP
      OUT     T3001Z1 K70
2907  LD      SM400  ; Alway on bit
      INC     Z1
2909  LD      T11  ; PLC_Alarm_Ready
      AND     Y16F  ; CART RIGHIT CYL LOCK SOL(PCO)
      AND     X13F  ; CART RIGHIT CYL LOCK CHECK_S6-2
      LD      L3001Z1
      ANI     L4003  ; Alarm Reset
      ANI     M3001Z1
      ORB
      MPS
      AND     T3001Z1
      OUT     L3166  ; CART RIGHT LOCK TIME OVER
      MPP
      OUT     T3001Z1 K70
2924  LD      SM400  ; Alway on bit
      INC     Z1
2926  LD      T11  ; PLC_Alarm_Ready
      ANI     Y16F  ; CART RIGHIT CYL LOCK SOL(PCO)
      ANI     X13F  ; CART RIGHIT CYL LOCK CHECK_S6-2
      LD      L3001Z1
      ANI     L4003  ; Alarm Reset
      ANI     M3001Z1
      ORB
      MPS
      AND     T3001Z1
      OUT     L3167  ; CART RIGHT UNLOCK TIME OVER
      MPP
      OUT     T3001Z1 K70
2941  LD      SM400  ; Alway on bit
      INC     Z1
2943  LD      T11  ; PLC_Alarm_Ready
      AND     X12D  ; CART UP POSITION CHECK SESOR(PCO
      AND     X139  ; CART DN POSITION CHECK SESOR_S12
      LD      L3001Z1
      ANI     L4003  ; Alarm Reset
      ANI     M3001Z1
      ORB
      MPS
      AND     T3001Z1
      OUT     L3168  ; CART LIFT SENSOR ERROR
      MPP
      OUT     T3001Z1 K10
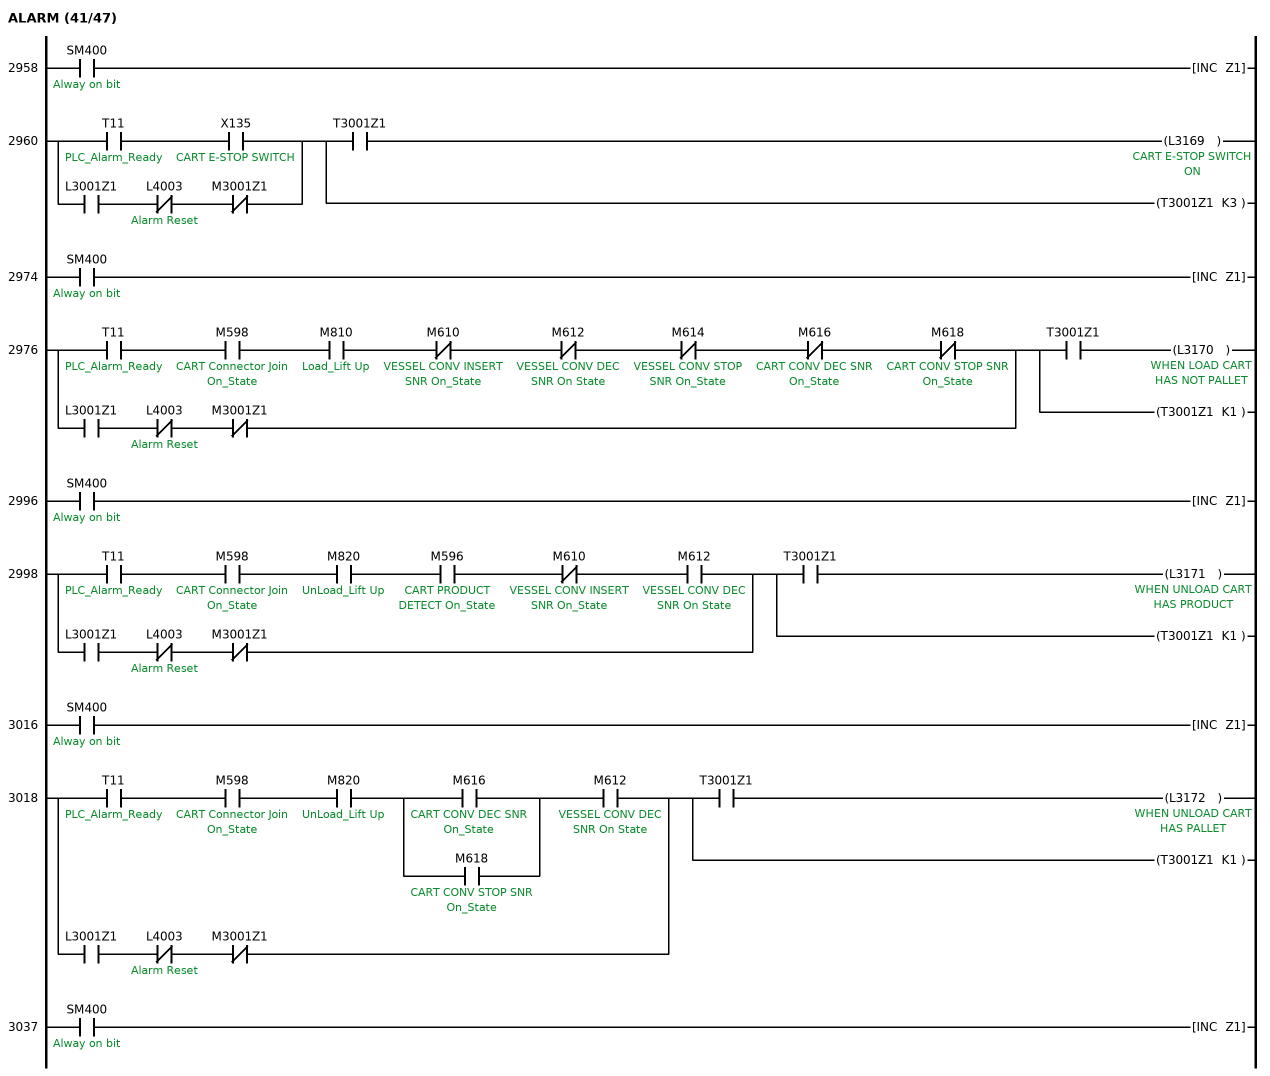
2958  LD      SM400  ; Alway on bit
      INC     Z1
2960  LD      T11  ; PLC_Alarm_Ready
      AND     X135  ; CART E-STOP SWITCH
      LD      L3001Z1
      ANI     L4003  ; Alarm Reset
      ANI     M3001Z1
      ORB
      MPS
      AND     T3001Z1
      OUT     L3169  ; CART E-STOP SWITCH ON
      MPP
      OUT     T3001Z1 K3
2974  LD      SM400  ; Alway on bit
      INC     Z1
2976  LD      T11  ; PLC_Alarm_Ready
      AND     M598  ; CART Connector Join On_State
      AND     M810  ; Load_Lift Up
      ANI     M610  ; VESSEL CONV INSERT SNR On_State
      ANI     M612  ; VESSEL CONV DEC SNR On State
      ANI     M614  ; VESSEL CONV STOP SNR On_State
      ANI     M616  ; CART CONV DEC SNR On_State
      ANI     M618  ; CART CONV STOP SNR On_State
      LD      L3001Z1
      ANI     L4003  ; Alarm Reset
      ANI     M3001Z1
      ORB
      MPS
      AND     T3001Z1
      OUT     L3170  ; WHEN LOAD CART HAS NOT PALLET
      MPP
      OUT     T3001Z1 K1
2996  LD      SM400  ; Alway on bit
      INC     Z1
2998  LD      T11  ; PLC_Alarm_Ready
      AND     M598  ; CART Connector Join On_State
      AND     M820  ; UnLoad_Lift Up
      AND     M596  ; CART PRODUCT DETECT On_State
      ANI     M610  ; VESSEL CONV INSERT SNR On_State
      AND     M612  ; VESSEL CONV DEC SNR On State
      LD      L3001Z1
      ANI     L4003  ; Alarm Reset
      ANI     M3001Z1
      ORB
      MPS
      AND     T3001Z1
      OUT     L3171  ; WHEN UNLOAD CART HAS PRODUCT
      MPP
      OUT     T3001Z1 K1
3016  LD      SM400  ; Alway on bit
      INC     Z1
3018  LD      T11  ; PLC_Alarm_Ready
      AND     M598  ; CART Connector Join On_State
      AND     M820  ; UnLoad_Lift Up
      LD      M616  ; CART CONV DEC SNR On_State
      OR      M618  ; CART CONV STOP SNR On_State
      ANB
      AND     M612  ; VESSEL CONV DEC SNR On State
      LD      L3001Z1
      ANI     L4003  ; Alarm Reset
      ANI     M3001Z1
      ORB
      MPS
      AND     T3001Z1
      OUT     L3172  ; WHEN UNLOAD CART HAS PALLET
      MPP
      OUT     T3001Z1 K1
3037  LD      SM400  ; Alway on bit
      INC     Z1
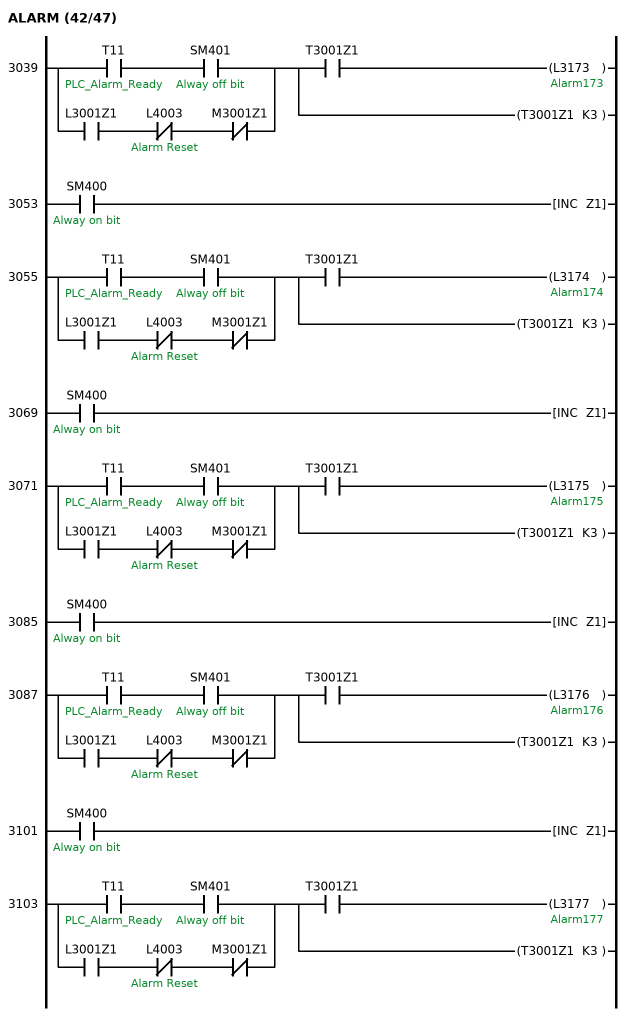
3039  LD      T11  ; PLC_Alarm_Ready
      AND     SM401  ; Alway off bit
      LD      L3001Z1
      ANI     L4003  ; Alarm Reset
      ANI     M3001Z1
      ORB
      MPS
      AND     T3001Z1
      OUT     L3173  ; Alarm173
      MPP
      OUT     T3001Z1 K3
3053  LD      SM400  ; Alway on bit
      INC     Z1
3055  LD      T11  ; PLC_Alarm_Ready
      AND     SM401  ; Alway off bit
      LD      L3001Z1
      ANI     L4003  ; Alarm Reset
      ANI     M3001Z1
      ORB
      MPS
      AND     T3001Z1
      OUT     L3174  ; Alarm174
      MPP
      OUT     T3001Z1 K3
3069  LD      SM400  ; Alway on bit
      INC     Z1
3071  LD      T11  ; PLC_Alarm_Ready
      AND     SM401  ; Alway off bit
      LD      L3001Z1
      ANI     L4003  ; Alarm Reset
      ANI     M3001Z1
      ORB
      MPS
      AND     T3001Z1
      OUT     L3175  ; Alarm175
      MPP
      OUT     T3001Z1 K3
3085  LD      SM400  ; Alway on bit
      INC     Z1
3087  LD      T11  ; PLC_Alarm_Ready
      AND     SM401  ; Alway off bit
      LD      L3001Z1
      ANI     L4003  ; Alarm Reset
      ANI     M3001Z1
      ORB
      MPS
      AND     T3001Z1
      OUT     L3176  ; Alarm176
      MPP
      OUT     T3001Z1 K3
3101  LD      SM400  ; Alway on bit
      INC     Z1
3103  LD      T11  ; PLC_Alarm_Ready
      AND     SM401  ; Alway off bit
      LD      L3001Z1
      ANI     L4003  ; Alarm Reset
      ANI     M3001Z1
      ORB
      MPS
      AND     T3001Z1
      OUT     L3177  ; Alarm177
      MPP
      OUT     T3001Z1 K3
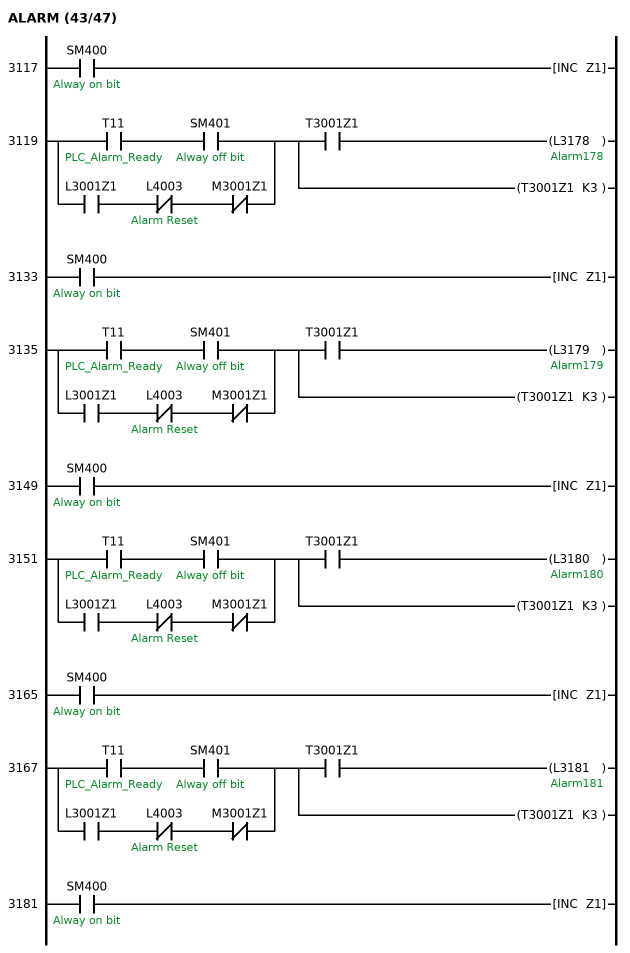
3117  LD      SM400  ; Alway on bit
      INC     Z1
3119  LD      T11  ; PLC_Alarm_Ready
      AND     SM401  ; Alway off bit
      LD      L3001Z1
      ANI     L4003  ; Alarm Reset
      ANI     M3001Z1
      ORB
      MPS
      AND     T3001Z1
      OUT     L3178  ; Alarm178
      MPP
      OUT     T3001Z1 K3
3133  LD      SM400  ; Alway on bit
      INC     Z1
3135  LD      T11  ; PLC_Alarm_Ready
      AND     SM401  ; Alway off bit
      LD      L3001Z1
      ANI     L4003  ; Alarm Reset
      ANI     M3001Z1
      ORB
      MPS
      AND     T3001Z1
      OUT     L3179  ; Alarm179
      MPP
      OUT     T3001Z1 K3
3149  LD      SM400  ; Alway on bit
      INC     Z1
3151  LD      T11  ; PLC_Alarm_Ready
      AND     SM401  ; Alway off bit
      LD      L3001Z1
      ANI     L4003  ; Alarm Reset
      ANI     M3001Z1
      ORB
      MPS
      AND     T3001Z1
      OUT     L3180  ; Alarm180
      MPP
      OUT     T3001Z1 K3
3165  LD      SM400  ; Alway on bit
      INC     Z1
3167  LD      T11  ; PLC_Alarm_Ready
      AND     SM401  ; Alway off bit
      LD      L3001Z1
      ANI     L4003  ; Alarm Reset
      ANI     M3001Z1
      ORB
      MPS
      AND     T3001Z1
      OUT     L3181  ; Alarm181
      MPP
      OUT     T3001Z1 K3
3181  LD      SM400  ; Alway on bit
      INC     Z1
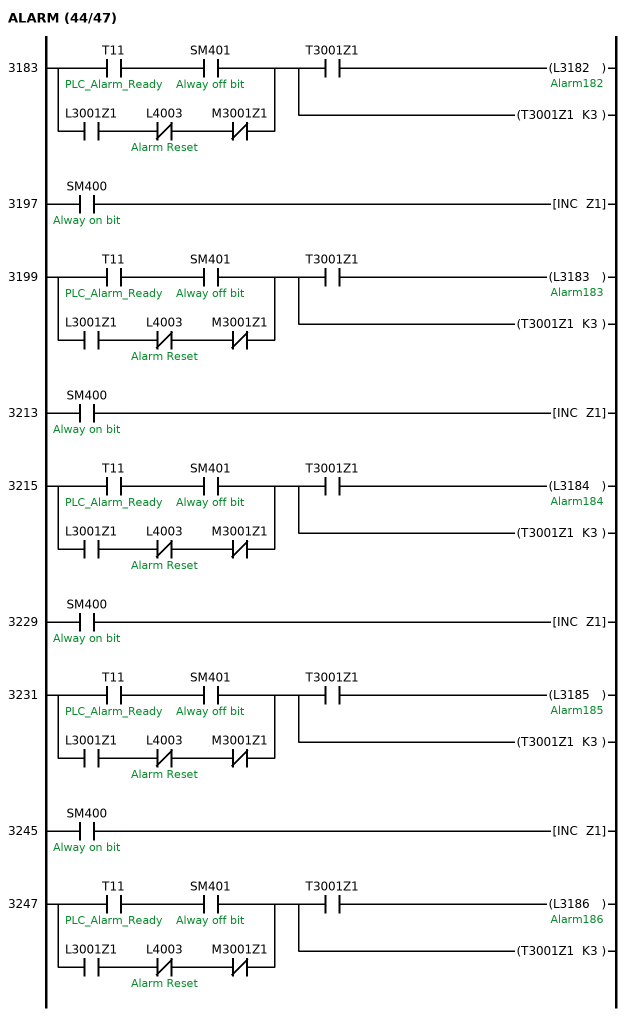
3183  LD      T11  ; PLC_Alarm_Ready
      AND     SM401  ; Alway off bit
      LD      L3001Z1
      ANI     L4003  ; Alarm Reset
      ANI     M3001Z1
      ORB
      MPS
      AND     T3001Z1
      OUT     L3182  ; Alarm182
      MPP
      OUT     T3001Z1 K3
3197  LD      SM400  ; Alway on bit
      INC     Z1
3199  LD      T11  ; PLC_Alarm_Ready
      AND     SM401  ; Alway off bit
      LD      L3001Z1
      ANI     L4003  ; Alarm Reset
      ANI     M3001Z1
      ORB
      MPS
      AND     T3001Z1
      OUT     L3183  ; Alarm183
      MPP
      OUT     T3001Z1 K3
3213  LD      SM400  ; Alway on bit
      INC     Z1
3215  LD      T11  ; PLC_Alarm_Ready
      AND     SM401  ; Alway off bit
      LD      L3001Z1
      ANI     L4003  ; Alarm Reset
      ANI     M3001Z1
      ORB
      MPS
      AND     T3001Z1
      OUT     L3184  ; Alarm184
      MPP
      OUT     T3001Z1 K3
3229  LD      SM400  ; Alway on bit
      INC     Z1
3231  LD      T11  ; PLC_Alarm_Ready
      AND     SM401  ; Alway off bit
      LD      L3001Z1
      ANI     L4003  ; Alarm Reset
      ANI     M3001Z1
      ORB
      MPS
      AND     T3001Z1
      OUT     L3185  ; Alarm185
      MPP
      OUT     T3001Z1 K3
3245  LD      SM400  ; Alway on bit
      INC     Z1
3247  LD      T11  ; PLC_Alarm_Ready
      AND     SM401  ; Alway off bit
      LD      L3001Z1
      ANI     L4003  ; Alarm Reset
      ANI     M3001Z1
      ORB
      MPS
      AND     T3001Z1
      OUT     L3186  ; Alarm186
      MPP
      OUT     T3001Z1 K3
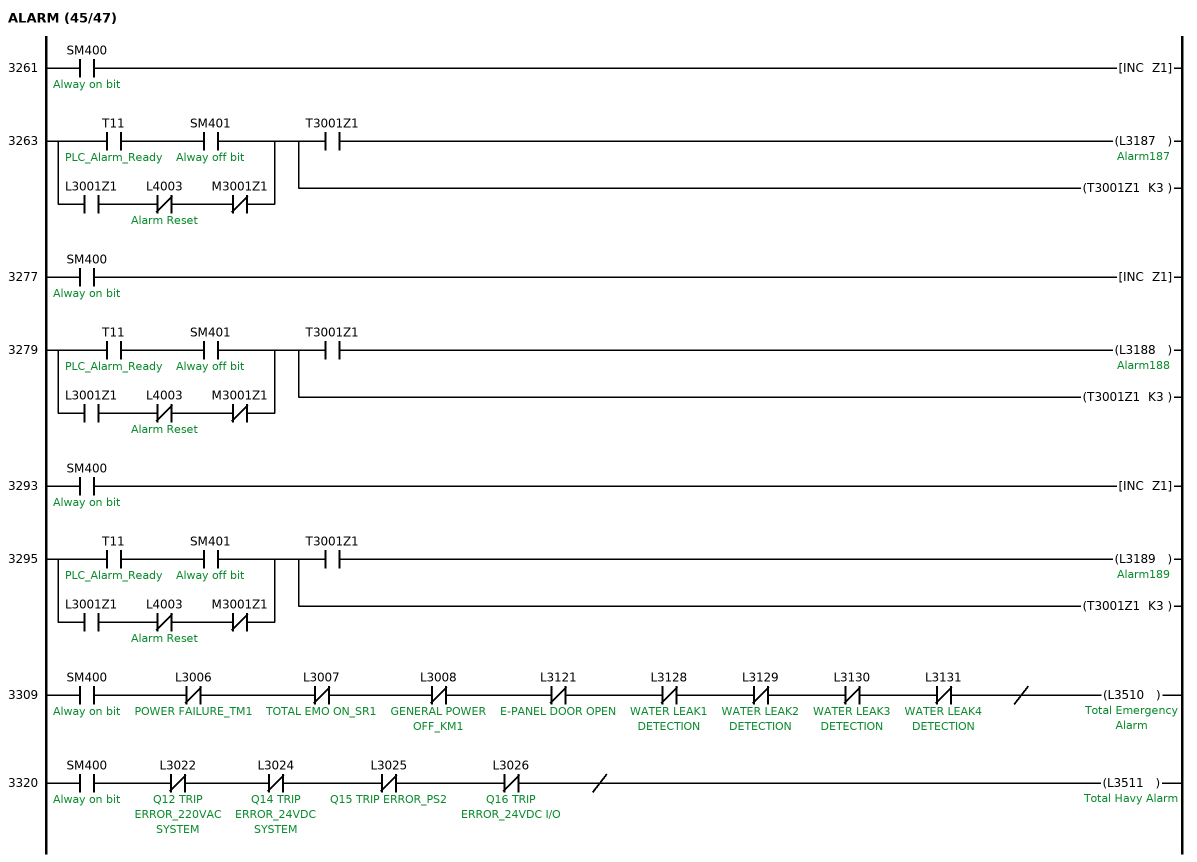
3261  LD      SM400  ; Alway on bit
      INC     Z1
3263  LD      T11  ; PLC_Alarm_Ready
      AND     SM401  ; Alway off bit
      LD      L3001Z1
      ANI     L4003  ; Alarm Reset
      ANI     M3001Z1
      ORB
      MPS
      AND     T3001Z1
      OUT     L3187  ; Alarm187
      MPP
      OUT     T3001Z1 K3
3277  LD      SM400  ; Alway on bit
      INC     Z1
3279  LD      T11  ; PLC_Alarm_Ready
      AND     SM401  ; Alway off bit
      LD      L3001Z1
      ANI     L4003  ; Alarm Reset
      ANI     M3001Z1
      ORB
      MPS
      AND     T3001Z1
      OUT     L3188  ; Alarm188
      MPP
      OUT     T3001Z1 K3
3293  LD      SM400  ; Alway on bit
      INC     Z1
3295  LD      T11  ; PLC_Alarm_Ready
      AND     SM401  ; Alway off bit
      LD      L3001Z1
      ANI     L4003  ; Alarm Reset
      ANI     M3001Z1
      ORB
      MPS
      AND     T3001Z1
      OUT     L3189  ; Alarm189
      MPP
      OUT     T3001Z1 K3
3309  LD      SM400  ; Alway on bit
      ANI     L3006  ; POWER FAILURE_TM1
      ANI     L3007  ; TOTAL EMO ON_SR1
      ANI     L3008  ; GENERAL POWER OFF_KM1
      ANI     L3121  ; E-PANEL DOOR OPEN
      ANI     L3128  ; WATER LEAK1 DETECTION
      ANI     L3129  ; WATER LEAK2 DETECTION
      ANI     L3130  ; WATER LEAK3 DETECTION
      ANI     L3131  ; WATER LEAK4 DETECTION
      INV
      OUT     L3510  ; Total Emergency Alarm
3320  LD      SM400  ; Alway on bit
      ANI     L3022  ; Q12 TRIP ERROR_220VAC SYSTEM
      ANI     L3024  ; Q14 TRIP ERROR_24VDC SYSTEM
      ANI     L3025  ; Q15 TRIP ERROR_PS2
      ANI     L3026  ; Q16 TRIP ERROR_24VDC I/O
      INV
      OUT     L3511  ; Total Havy Alarm
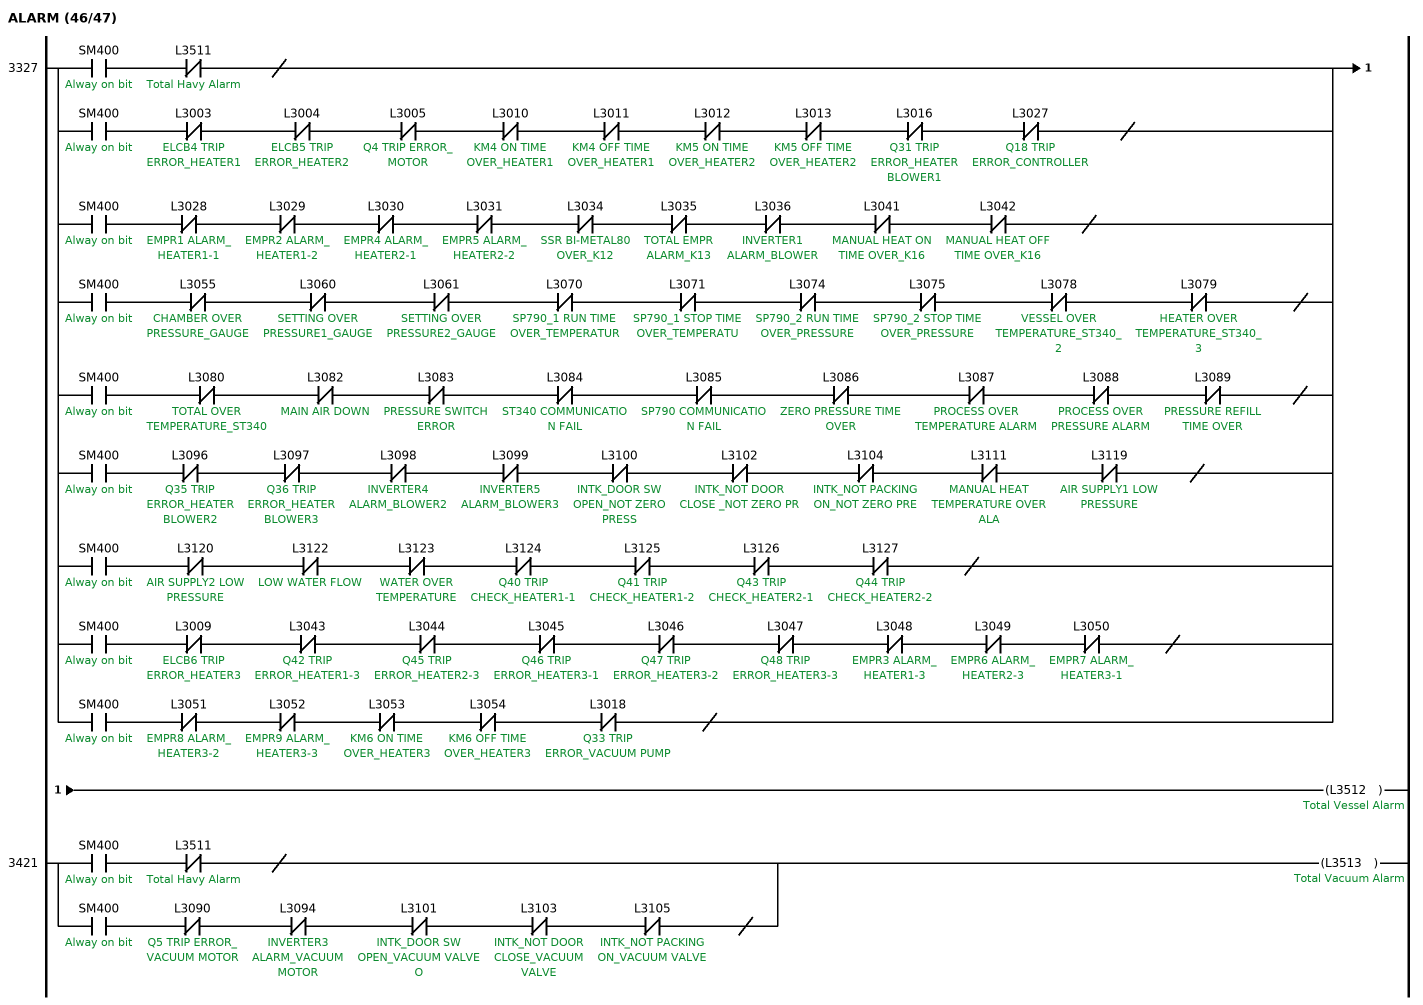
3327  LD      SM400  ; Alway on bit
      ANI     L3511  ; Total Havy Alarm
      INV
      LD      SM400  ; Alway on bit
      ANI     L3003  ; ELCB4 TRIP ERROR_HEATER1
      ANI     L3004  ; ELCB5 TRIP ERROR_HEATER2
      ANI     L3005  ; Q4 TRIP ERROR_MOTOR
      ANI     L3010  ; KM4 ON TIME OVER_HEATER1
      ANI     L3011  ; KM4 OFF TIME OVER_HEATER1
      ANI     L3012  ; KM5 ON TIME OVER_HEATER2
      ANI     L3013  ; KM5 OFF TIME OVER_HEATER2
      ANI     L3016  ; Q31 TRIP ERROR_HEATER BLOWER1
      ANI     L3027  ; Q18 TRIP ERROR_CONTROLLER
      INV
      ORB
      LD      SM400  ; Alway on bit
      ANI     L3028  ; EMPR1 ALARM_HEATER1-1
      ANI     L3029  ; EMPR2 ALARM_HEATER1-2
      ANI     L3030  ; EMPR4 ALARM_HEATER2-1
      ANI     L3031  ; EMPR5 ALARM_HEATER2-2
      ANI     L3034  ; SSR BI-METAL80 OVER_K12
      ANI     L3035  ; TOTAL EMPR ALARM_K13
      ANI     L3036  ; INVERTER1 ALARM_BLOWER
      ANI     L3041  ; MANUAL HEAT ON TIME OVER_K16
      ANI     L3042  ; MANUAL HEAT OFF TIME OVER_K16
      INV
      ORB
      LD      SM400  ; Alway on bit
      ANI     L3055  ; CHAMBER OVER PRESSURE_GAUGE
      ANI     L3060  ; SETTING OVER PRESSURE1_GAUGE
      ANI     L3061  ; SETTING OVER PRESSURE2_GAUGE
      ANI     L3070  ; SP790_1 RUN TIME OVER_TEMPERATUR
      ANI     L3071  ; SP790_1 STOP TIME OVER_TEMPERATU
      ANI     L3074  ; SP790_2 RUN TIME OVER_PRESSURE
      ANI     L3075  ; SP790_2 STOP TIME OVER_PRESSURE
      ANI     L3078  ; VESSEL OVER TEMPERATURE_ST340_2
      ANI     L3079  ; HEATER OVER TEMPERATURE_ST340_3
      INV
      ORB
      LD      SM400  ; Alway on bit
      ANI     L3080  ; TOTAL OVER TEMPERATURE_ST340
      ANI     L3082  ; MAIN AIR DOWN
      ANI     L3083  ; PRESSURE SWITCH ERROR
      ANI     L3084  ; ST340 COMMUNICATION FAIL
      ANI     L3085  ; SP790 COMMUNICATION FAIL
      ANI     L3086  ; ZERO PRESSURE TIME OVER
      ANI     L3087  ; PROCESS OVER TEMPERATURE ALARM
      ANI     L3088  ; PROCESS OVER PRESSURE ALARM
      ANI     L3089  ; PRESSURE REFILL TIME OVER
      INV
      ORB
      LD      SM400  ; Alway on bit
      ANI     L3096  ; Q35 TRIP ERROR_HEATER BLOWER2
      ANI     L3097  ; Q36 TRIP ERROR_HEATER BLOWER3
      ANI     L3098  ; INVERTER4 ALARM_BLOWER2
      ANI     L3099  ; INVERTER5 ALARM_BLOWER3
      ANI     L3100  ; INTK_DOOR SW OPEN_NOT ZERO PRESS
      ANI     L3102  ; INTK_NOT DOOR CLOSE _NOT ZERO PR
      ANI     L3104  ; INTK_NOT PACKING ON_NOT ZERO PRE
      ANI     L3111  ; MANUAL HEAT TEMPERATURE OVER ALA
      ANI     L3119  ; AIR SUPPLY1 LOW PRESSURE
      INV
      ORB
      LD      SM400  ; Alway on bit
      ANI     L3120  ; AIR SUPPLY2 LOW PRESSURE
      ANI     L3122  ; LOW WATER FLOW
      ANI     L3123  ; WATER OVER TEMPERATURE
      ANI     L3124  ; Q40 TRIP CHECK_HEATER1-1
      ANI     L3125  ; Q41 TRIP CHECK_HEATER1-2
      ANI     L3126  ; Q43 TRIP CHECK_HEATER2-1
      ANI     L3127  ; Q44 TRIP CHECK_HEATER2-2
      INV
      ORB
      LD      SM400  ; Alway on bit
      ANI     L3009  ; ELCB6 TRIP ERROR_HEATER3
      ANI     L3043  ; Q42 TRIP ERROR_HEATER1-3
      ANI     L3044  ; Q45 TRIP ERROR_HEATER2-3
      ANI     L3045  ; Q46 TRIP ERROR_HEATER3-1
      ANI     L3046  ; Q47 TRIP ERROR_HEATER3-2
      ANI     L3047  ; Q48 TRIP ERROR_HEATER3-3
      ANI     L3048  ; EMPR3 ALARM_HEATER1-3
      ANI     L3049  ; EMPR6 ALARM_HEATER2-3
      ANI     L3050  ; EMPR7 ALARM_HEATER3-1
      INV
      ORB
      LD      SM400  ; Alway on bit
      ANI     L3051  ; EMPR8 ALARM_HEATER3-2
      ANI     L3052  ; EMPR9 ALARM_HEATER3-3
      ANI     L3053  ; KM6 ON TIME OVER_HEATER3
      ANI     L3054  ; KM6 OFF TIME OVER_HEATER3
      ANI     L3018  ; Q33 TRIP ERROR_VACUUM PUMP
      INV
      ORB
      OUT     L3512  ; Total Vessel Alarm
3421  LD      SM400  ; Alway on bit
      ANI     L3511  ; Total Havy Alarm
      INV
      LD      SM400  ; Alway on bit
      ANI     L3090  ; Q5 TRIP ERROR_VACUUM MOTOR
      ANI     L3094  ; INVERTER3 ALARM_VACUUM MOTOR
      ANI     L3101  ; INTK_DOOR SW OPEN_VACUUM VALVE O
      ANI     L3103  ; INTK_NOT DOOR CLOSE_VACUUM VALVE
      ANI     L3105  ; INTK_NOT PACKING ON_VACUUM VALVE
      INV
      ORB
      OUT     L3513  ; Total Vacuum Alarm
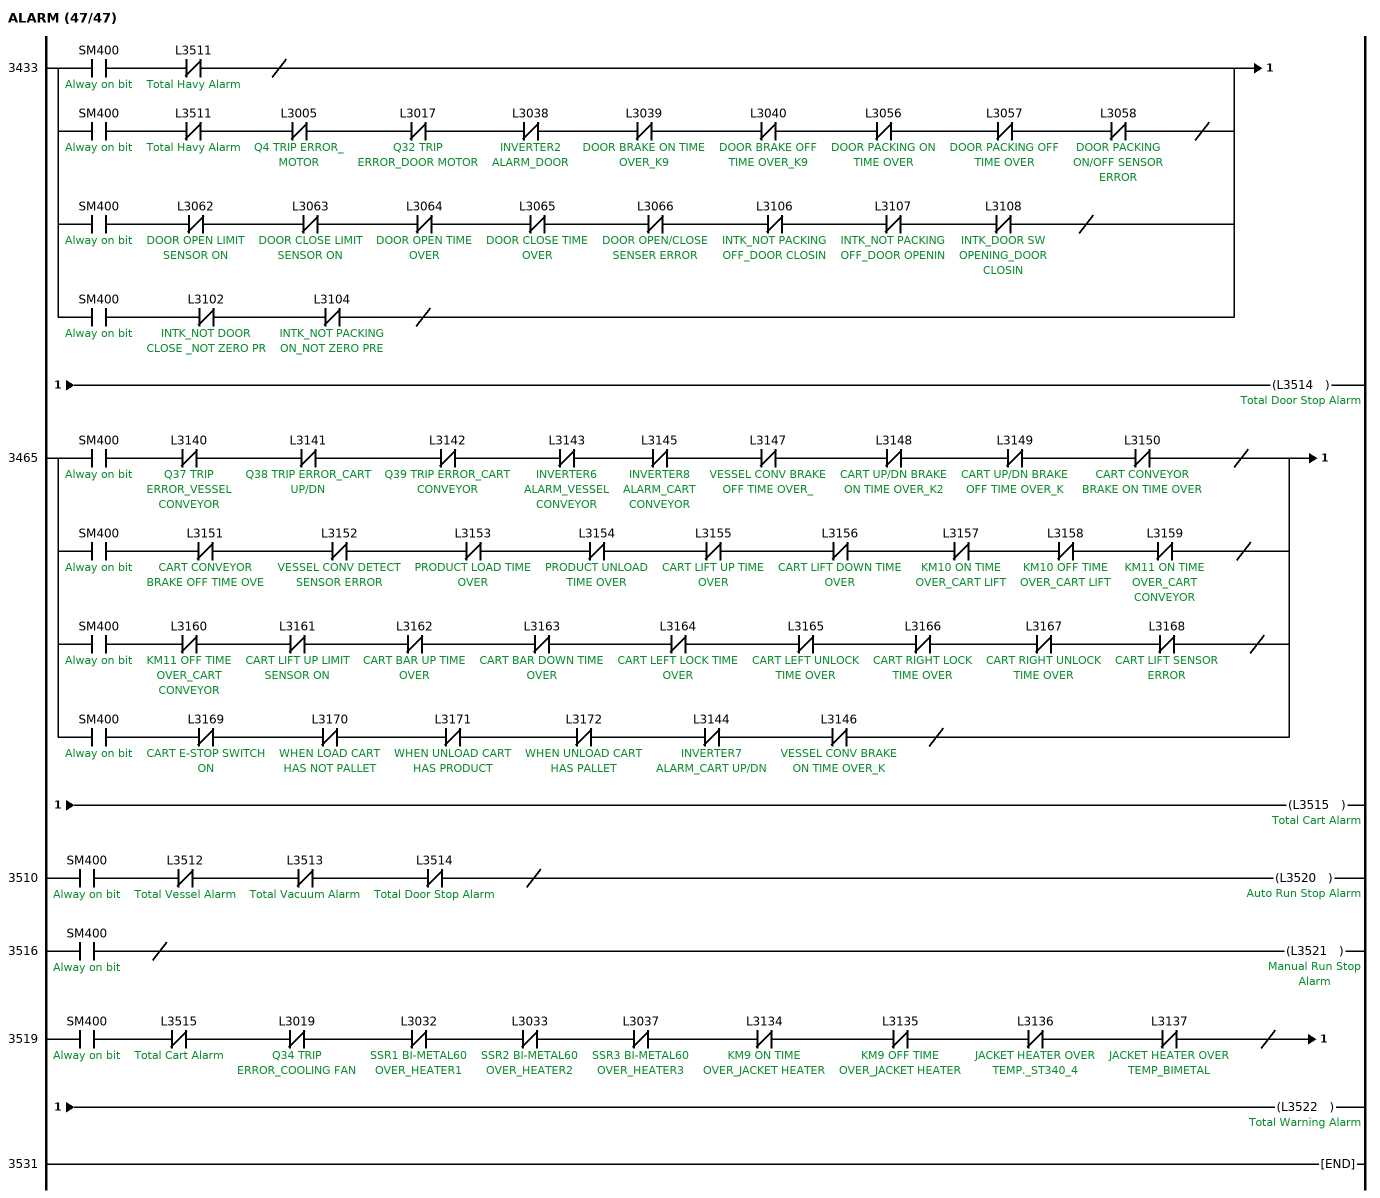
3433  LD      SM400  ; Alway on bit
      ANI     L3511  ; Total Havy Alarm
      INV
      LD      SM400  ; Alway on bit
      ANI     L3511  ; Total Havy Alarm
      ANI     L3005  ; Q4 TRIP ERROR_MOTOR
      ANI     L3017  ; Q32 TRIP ERROR_DOOR MOTOR
      ANI     L3038  ; INVERTER2 ALARM_DOOR
      ANI     L3039  ; DOOR BRAKE ON TIME OVER_K9
      ANI     L3040  ; DOOR BRAKE OFF TIME OVER_K9
      ANI     L3056  ; DOOR PACKING ON TIME OVER
      ANI     L3057  ; DOOR PACKING OFF TIME OVER
      ANI     L3058  ; DOOR PACKING ON/OFF SENSOR ERROR
      INV
      ORB
      LD      SM400  ; Alway on bit
      ANI     L3062  ; DOOR OPEN LIMIT SENSOR ON
      ANI     L3063  ; DOOR CLOSE LIMIT SENSOR ON
      ANI     L3064  ; DOOR OPEN TIME OVER
      ANI     L3065  ; DOOR CLOSE TIME OVER
      ANI     L3066  ; DOOR OPEN/CLOSE SENSER ERROR
      ANI     L3106  ; INTK_NOT PACKING OFF_DOOR CLOSIN
      ANI     L3107  ; INTK_NOT PACKING OFF_DOOR OPENIN
      ANI     L3108  ; INTK_DOOR SW OPENING_DOOR CLOSIN
      INV
      ORB
      LD      SM400  ; Alway on bit
      ANI     L3102  ; INTK_NOT DOOR CLOSE _NOT ZERO PR
      ANI     L3104  ; INTK_NOT PACKING ON_NOT ZERO PRE
      INV
      ORB
      OUT     L3514  ; Total Door Stop Alarm
3465  LD      SM400  ; Alway on bit
      ANI     L3140  ; Q37 TRIP ERROR_VESSEL CONVEYOR
      ANI     L3141  ; Q38 TRIP ERROR_CART UP/DN
      ANI     L3142  ; Q39 TRIP ERROR_CART CONVEYOR
      ANI     L3143  ; INVERTER6 ALARM_VESSEL CONVEYOR
      ANI     L3145  ; INVERTER8 ALARM_CART CONVEYOR
      ANI     L3147  ; VESSEL CONV BRAKE OFF TIME OVER_
      ANI     L3148  ; CART UP/DN BRAKE ON TIME OVER_K2
      ANI     L3149  ; CART UP/DN BRAKE OFF TIME OVER_K
      ANI     L3150  ; CART CONVEYOR BRAKE ON TIME OVER
      INV
      LD      SM400  ; Alway on bit
      ANI     L3151  ; CART CONVEYOR BRAKE OFF TIME OVE
      ANI     L3152  ; VESSEL CONV DETECT SENSOR ERROR
      ANI     L3153  ; PRODUCT LOAD TIME OVER
      ANI     L3154  ; PRODUCT UNLOAD TIME OVER
      ANI     L3155  ; CART LIFT UP TIME OVER
      ANI     L3156  ; CART LIFT DOWN TIME OVER
      ANI     L3157  ; KM10 ON TIME OVER_CART LIFT
      ANI     L3158  ; KM10 OFF TIME OVER_CART LIFT
      ANI     L3159  ; KM11 ON TIME OVER_CART CONVEYOR
      INV
      ORB
      LD      SM400  ; Alway on bit
      ANI     L3160  ; KM11 OFF TIME OVER_CART CONVEYOR
      ANI     L3161  ; CART LIFT UP LIMIT SENSOR ON
      ANI     L3162  ; CART BAR UP TIME OVER
      ANI     L3163  ; CART BAR DOWN TIME OVER
      ANI     L3164  ; CART LEFT LOCK TIME OVER
      ANI     L3165  ; CART LEFT UNLOCK TIME OVER
      ANI     L3166  ; CART RIGHT LOCK TIME OVER
      ANI     L3167  ; CART RIGHT UNLOCK TIME OVER
      ANI     L3168  ; CART LIFT SENSOR ERROR
      INV
      ORB
      LD      SM400  ; Alway on bit
      ANI     L3169  ; CART E-STOP SWITCH ON
      ANI     L3170  ; WHEN LOAD CART HAS NOT PALLET
      ANI     L3171  ; WHEN UNLOAD CART HAS PRODUCT
      ANI     L3172  ; WHEN UNLOAD CART HAS PALLET
      ANI     L3144  ; INVERTER7 ALARM_CART UP/DN
      ANI     L3146  ; VESSEL CONV BRAKE ON TIME OVER_K
      INV
      ORB
      OUT     L3515  ; Total Cart Alarm
3510  LD      SM400  ; Alway on bit
      ANI     L3512  ; Total Vessel Alarm
      ANI     L3513  ; Total Vacuum Alarm
      ANI     L3514  ; Total Door Stop Alarm
      INV
      OUT     L3520  ; Auto Run Stop Alarm
3516  LD      SM400  ; Alway on bit
      INV
      OUT     L3521  ; Manual Run Stop Alarm
3519  LD      SM400  ; Alway on bit
      ANI     L3515  ; Total Cart Alarm
      ANI     L3019  ; Q34 TRIP ERROR_COOLING FAN
      ANI     L3032  ; SSR1 BI-METAL60 OVER_HEATER1
      ANI     L3033  ; SSR2 BI-METAL60 OVER_HEATER2
      ANI     L3037  ; SSR3 BI-METAL60 OVER_HEATER3
      ANI     L3134  ; KM9 ON TIME OVER_JACKET HEATER
      ANI     L3135  ; KM9 OFF TIME OVER_JACKET HEATER
      ANI     L3136  ; JACKET HEATER OVER TEMP._ST340_4
      ANI     L3137  ; JACKET HEATER OVER TEMP_BIMETAL
      INV
      OUT     L3522  ; Total Warning Alarm
3531  END
END_PROGRAM
